KUKA KRL program: EPS_2_251455_MH12A_A_20251003045058.src

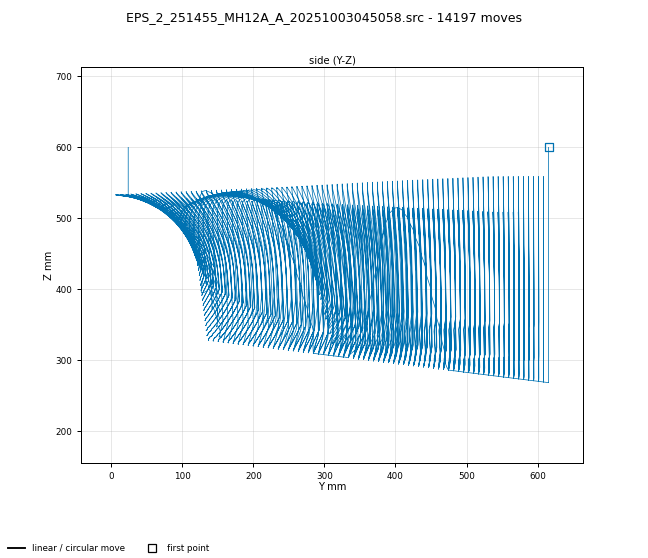
[picture p0: tool path of EPS_2_251455_MH12A_A_20251003045058.src, 14197 of 14199 moves have a stored position in this frame; points joined in program order, loops and branches not executed]
&ACCESS RVP
&REL 4
&COMMENT QRS 19112012
&PARAM EDITMASK = *
DEF PART()
EXT BAS (BAS_COMMAND :IN,REAL :IN )
INT I
BAS (#INITMOV,0 )

;KUKA QRS Post kuka4.cps  Date:22-06-2017 !

File_ID=2868

QRS_PRE_INIT()

;Init var - Until changes are made in qrs_pre_init
Outlet_Square_prg=0
Inlet_1_Square_prg=0
Inlet_2_Square_prg=0
Inlet_3_Square_prg=0
Inlet_4_Square_prg=0
Inlet_5_Square_prg=0

Outlet_1={X 0.000, Y 535.490, Z 458.500, B 0.000, E1 0.000 }
Inlet_1={X 0.000, Y 539.060, Z 408.500, B 0.000, E1 180.000 }
Inlet_2={X 0.000, Y 539.060, Z 408.500, B 0.000, E1 270.000 }
Outlet_1_type=201
Inlet_1_type=201
Inlet_2_type=201
;QRS#1=Sidecore dimensions
;QRS#2=200-8" PVC SDR 35
;QRS#3=200-8" PVC SDR 35
;QRS#4=200-8" PVC SDR 35
;QRS#5=
;QRS#6=
;QRS#7=
;QRS#8=
;QRS#9=12-08 PSX
;QRS#10=12-08 PSX
;QRS#11=12-08 PSX
;QRS#12=
;QRS#13=
;QRS#14=
;QRS#15=
;QRS#16=1220x127x838 2,75'
;QRS#17=EPS Height
;QRS#18=559
;QRS#19=*
;QRS#20= UPDATED VERSION 22-06-2017
;QRS#21=*
Outlet_Square=0100
Inlet_1_Square=0100
Inlet_2_Square=0100
Inlet_3_Square=0
Inlet_4_Square=0
Inlet_5_Square=0
Mill_Square=1
Outlet_Square_Prg=204
Inlet_1_Square_prg=204
Inlet_2_Square_prg=204

QRS_INIT()

$ADVANCE=5

; T1
PTP {E1 173.612,E2 173.612}
PTP {X 0,Y 615.502,A -85,B 0,C 180,E1 173.612,E2 173.612,E3 0,E4 0,E5 0,E6 0}
QRS_SPEED_INIT()
LIN {X 0,Y 615.502,Z 600,A -85,B 0,C 180,E1 173.612,E2 173.612,E3 0,E4 0,E5 0,E6 0} C_VEL
LIN {X 0,Y 615.502,Z 278.875,A -85,B 0,C 180,E1 173.612,E2 173.612} C_VEL
LIN {X 0,Y 615.502,Z 270.697,A -85,B 0,C 180,E1 173.612,E2 173.612} C_VEL
LIN {X 0,Y 615.472,Z 268.697,A -85,B 0,C 180,E1 173.426,E2 173.426} C_VEL
LIN {X 0,Y 615.422,Z 268.698,A -85,B 0,C 180,E1 170.8,E2 170.8} C_VEL
LIN {X 0,Y 615.459,Z 268.699,A -85,B 0,C 180,E1 168.139,E2 168.139} C_VEL
LIN {X 0,Y 615.46,Z 268.695,A -85,B 0,C 180,E1 165.45,E2 165.45} C_VEL
LIN {X 0,Y 615.453,Z 268.695,A -85,B 0,C 180,E1 163.412,E2 163.412} C_VEL
LIN {X 0,Y 615.446,Z 268.695,A -85,B 0,C 180,E1 161.353,E2 161.353} C_VEL
LIN {X 0,Y 615.437,Z 268.695,A -85,B 0,C 180,E1 159.267,E2 159.267} C_VEL
LIN {X 0,Y 615.434,Z 268.695,A -85,B 0,C 180,E1 157.153,E2 157.153} C_VEL
LIN {X 0,Y 615.433,Z 268.696,A -85,B 0,C 180,E1 155.006,E2 155.006} C_VEL
LIN {X 0,Y 615.493,Z 268.695,A -85,B 0,C 180,E1 152.085,E2 152.085} C_VEL
LIN {X 0,Y 615.478,Z 268.69,A -85,B 0,C 180,E1 149.839,E2 149.839} C_VEL
LIN {X 0,Y 615.448,Z 268.692,A -85,B 0,C 180,E1 147.54,E2 147.54} C_VEL
LIN {X 0,Y 615.44,Z 268.695,A -85,B 0,C 180,E1 145.182,E2 145.182} C_VEL
LIN {X 0,Y 615.469,Z 268.698,A -85,B 0,C 180,E1 142.756,E2 142.756} C_VEL
LIN {X 0,Y 615.47,Z 268.689,A -85,B 0,C 180,E1 139.912,E2 139.912} C_VEL
LIN {X 0,Y 615.449,Z 268.692,A -85,B 0,C 180,E1 137.643,E2 137.643} C_VEL
LIN {X 0,Y 615.469,Z 268.699,A -85,B 0,C 180,E1 134.929,E2 134.929} C_VEL
LIN {X 0,Y 615.475,Z 268.688,A -85,B 0,C 180,E1 132.079,E2 132.079} C_VEL
LIN {X 0,Y 615.452,Z 268.691,A -85,B 0,C 180,E1 129.752,E2 129.752} C_VEL
LIN {X 0,Y 615.485,Z 268.703,A -85,B 0,C 180,E1 126.936,E2 126.936} C_VEL
LIN {X 0,Y 615.459,Z 268.689,A -85,B 0,C 180,E1 124.023,E2 124.023} C_VEL
LIN {X 0,Y 615.455,Z 268.693,A -85,B 0,C 180,E1 121.686,E2 121.686} C_VEL
LIN {X 0,Y 615.47,Z 268.697,A -85,B 0,C 180,E1 119.406,E2 119.406} C_VEL
LIN {X 0,Y 615.482,Z 268.685,A -85,B 0,C 180,E1 116.443,E2 116.443} C_VEL
LIN {X 0,Y 615.46,Z 268.69,A -85,B 0,C 180,E1 114.002,E2 114.002} C_VEL
LIN {X 0,Y 615.486,Z 268.699,A -85,B 0,C 180,E1 111.431,E2 111.431} C_VEL
LIN {X 0,Y 615.486,Z 268.684,A -85,B 0,C 180,E1 108.603,E2 108.603} C_VEL
LIN {X 0,Y 615.464,Z 268.876,A -85,B 0,C 180,E1 107.957,E2 107.957} C_VEL
LIN {X 0,Y 615.478,Z 284.471,A -85,B 0,C 180,E1 105.225,E2 105.225} C_VEL
LIN {X 0,Y 615.49,Z 298.338,A -85,B 0,C 180,E1 102.823,E2 102.823} C_VEL
LIN {X 0,Y 615.481,Z 405.834,A -85,B 0,C 180,E1 101.526,E2 101.526} C_VEL
LIN {X 0,Y 615.475,Z 418.769,A -85,B 0,C 180,E1 101.234,E2 101.234} C_VEL
LIN {X 0,Y 615.492,Z 430.613,A -85,B 0,C 180,E1 100.842,E2 100.842} C_VEL
LIN {X 0,Y 615.48,Z 441.583,A -85,B 0,C 180,E1 100.36,E2 100.36} C_VEL
LIN {X 0,Y 615.493,Z 453.315,A -85,B 0,C 180,E1 99.695,E2 99.695} C_VEL
LIN {X 0,Y 615.499,Z 463.777,A -85,B 0,C 180,E1 98.949,E2 98.949} C_VEL
LIN {X 0,Y 615.498,Z 472.338,A -85,B 0,C 180,E1 98.205,E2 98.205} C_VEL
LIN {X 0,Y 615.497,Z 480.215,A -85,B 0,C 180,E1 97.38,E2 97.38} C_VEL
LIN {X 0,Y 615.497,Z 487.903,A -85,B 0,C 180,E1 96.391,E2 96.391} C_VEL
LIN {X 0,Y 615.497,Z 494.962,A -85,B 0,C 180,E1 95.24,E2 95.24} C_VEL
LIN {X 0,Y 615.494,Z 499.661,A -85,B 0,C 180,E1 94.256,E2 94.256} C_VEL
LIN {X 0,Y 615.494,Z 503.257,A -85,B 0,C 180,E1 93.272,E2 93.272} C_VEL
LIN {X 0,Y 615.496,Z 505.116,A -85,B 0,C 180,E1 92.617,E2 92.617} C_VEL
LIN {X 0,Y 615.5,Z 506.534,A -85,B 0,C 180,E1 91.962,E2 91.962} C_VEL
LIN {X 0,Y 615.496,Z 508.142,A -85,B 0,C 180,E1 90.654,E2 90.654} C_VEL
LIN {X 0,Y 615.495,Z 508.384,A -85,B 0,C 180,E1 89.999,E2 89.999} C_VEL
LIN {X 0,Y 615.495,Z 508.205,A -85,B 0,C 180,E1 89.345,E2 89.345} C_VEL
LIN {X 0,Y 615.5,Z 506.681,A -85,B 0,C 180,E1 88.036,E2 88.036} C_VEL
LIN {X 0,Y 615.498,Z 505.34,A -85,B 0,C 180,E1 87.382,E2 87.382} C_VEL
LIN {X 0,Y 615.496,Z 502.492,A -85,B 0,C 180,E1 86.399,E2 86.399} C_VEL
LIN {X 0,Y 615.498,Z 498.632,A -85,B 0,C 180,E1 85.415,E2 85.415} C_VEL
LIN {X 0,Y 615.498,Z 493.648,A -85,B 0,C 180,E1 84.43,E2 84.43} C_VEL
LIN {X 0,Y 615.496,Z 487.208,A -85,B 0,C 180,E1 83.418,E2 83.418} C_VEL
LIN {X 0,Y 615.497,Z 479.531,A -85,B 0,C 180,E1 82.454,E2 82.454} C_VEL
LIN {X 0,Y 615.498,Z 469.752,A -85,B 0,C 180,E1 81.463,E2 81.463} C_VEL
LIN {X 0,Y 615.498,Z 459.484,A -85,B 0,C 180,E1 80.635,E2 80.635} C_VEL
LIN {X 0,Y 615.483,Z 447.921,A -85,B 0,C 180,E1 79.888,E2 79.888} C_VEL
LIN {X 0,Y 615.495,Z 436.069,A -85,B 0,C 180,E1 79.293,E2 79.293} C_VEL
LIN {X 0,Y 615.475,Z 423.143,A -85,B 0,C 180,E1 78.806,E2 78.806} C_VEL
LIN {X 0,Y 615.481,Z 410.534,A -85,B 0,C 180,E1 78.473,E2 78.473} C_VEL
LIN {X 0,Y 615.49,Z 397.384,A -85,B 0,C 180,E1 78.264,E2 78.264} C_VEL
LIN {X 0,Y 615.49,Z 298.366,A -85,B 0,C 180,E1 77.092,E2 77.092} C_VEL
LIN {X 0,Y 615.48,Z 283.028,A -85,B 0,C 180,E1 74.434,E2 74.434} C_VEL
LIN {X 0,Y 615.468,Z 268.69,A -85,B 0,C 180,E1 71.901,E2 71.901} C_VEL
LIN {X 0,Y 615.488,Z 268.684,A -85,B 0,C 180,E1 69.269,E2 69.269} C_VEL
LIN {X 0,Y 615.48,Z 268.699,A -85,B 0,C 180,E1 66.443,E2 66.443} C_VEL
LIN {X 0,Y 615.484,Z 268.683,A -85,B 0,C 180,E1 63.555,E2 63.555} C_VEL
LIN {X 0,Y 615.485,Z 268.7,A -85,B 0,C 180,E1 60.593,E2 60.593} C_VEL
LIN {X 0,Y 615.487,Z 268.683,A -85,B 0,C 180,E1 57.67,E2 57.67} C_VEL
LIN {X 0,Y 615.486,Z 268.69,A -85,B 0,C 180,E1 55.184,E2 55.184} C_VEL
LIN {X 0,Y 615.49,Z 268.7,A -85,B 0,C 180,E1 52.758,E2 52.758} C_VEL
LIN {X 0,Y 615.477,Z 268.685,A -85,B 0,C 180,E1 49.913,E2 49.913} C_VEL
LIN {X 0,Y 615.488,Z 268.702,A -85,B 0,C 180,E1 46.953,E2 46.953} C_VEL
LIN {X 0,Y 615.47,Z 268.687,A -85,B 0,C 180,E1 44.151,E2 44.151} C_VEL
LIN {X 0,Y 615.484,Z 268.689,A -85,B 0,C 180,E1 41.474,E2 41.474} C_VEL
LIN {X 0,Y 615.486,Z 268.698,A -85,B 0,C 180,E1 38.905,E2 38.905} C_VEL
LIN {X 0,Y 615.468,Z 268.689,A -85,B 0,C 180,E1 36.426,E2 36.426} C_VEL
LIN {X 0,Y 615.486,Z 268.691,A -85,B 0,C 180,E1 33.533,E2 33.533} C_VEL
LIN {X 0,Y 615.474,Z 268.696,A -85,B 0,C 180,E1 30.921,E2 30.921} C_VEL
LIN {X 0,Y 615.47,Z 268.687,A -85,B 0,C 180,E1 28.447,E2 28.447} C_VEL
LIN {X 0,Y 615.487,Z 268.693,A -85,B 0,C 180,E1 25.568,E2 25.568} C_VEL
LIN {X 0,Y 615.467,Z 268.693,A -85,B 0,C 180,E1 22.845,E2 22.845} C_VEL
LIN {X 0,Y 615.492,Z 268.684,A -85,B 0,C 180,E1 20.033,E2 20.033} C_VEL
LIN {X 0,Y 615.484,Z 268.869,A -85,B 0,C 180,E1 17.957,E2 17.957} C_VEL
LIN {X 0,Y 615.454,Z 284.469,A -85,B 0,C 180,E1 15.227,E2 15.227} C_VEL
LIN {X 0,Y 615.478,Z 298.626,A -85,B 0,C 180,E1 12.803,E2 12.803} C_VEL
LIN {X 0,Y 615.484,Z 404.641,A -85,B 0,C 180,E1 11.548,E2 11.548} C_VEL
LIN {X 0,Y 615.493,Z 417.22,A -85,B 0,C 180,E1 11.276,E2 11.276} C_VEL
LIN {X 0,Y 615.493,Z 430.577,A -85,B 0,C 180,E1 10.843,E2 10.843} C_VEL
LIN {X 0,Y 615.492,Z 441.564,A -85,B 0,C 180,E1 10.361,E2 10.361} C_VEL
LIN {X 0,Y 615.479,Z 453.305,A -85,B 0,C 180,E1 9.696,E2 9.696} C_VEL
LIN {X 0,Y 615.499,Z 463.767,A -85,B 0,C 180,E1 8.95,E2 8.95} C_VEL
LIN {X 0,Y 615.498,Z 472.33,A -85,B 0,C 180,E1 8.206,E2 8.206} C_VEL
LIN {X 0,Y 615.497,Z 480.209,A -85,B 0,C 180,E1 7.38,E2 7.38} C_VEL
LIN {X 0,Y 615.497,Z 487.898,A -85,B 0,C 180,E1 6.392,E2 6.392} C_VEL
LIN {X 0,Y 615.498,Z 494.958,A -85,B 0,C 180,E1 5.241,E2 5.241} C_VEL
LIN {X 0,Y 615.493,Z 499.658,A -85,B 0,C 180,E1 4.256,E2 4.256} C_VEL
LIN {X 0,Y 615.496,Z 503.254,A -85,B 0,C 180,E1 3.273,E2 3.273} C_VEL
LIN {X 0,Y 615.496,Z 505.115,A -85,B 0,C 180,E1 2.618,E2 2.618} C_VEL
LIN {X 0,Y 615.497,Z 506.533,A -85,B 0,C 180,E1 1.963,E2 1.963} C_VEL
LIN {X 0,Y 615.496,Z 508.141,A -85,B 0,C 180,E1 0.654,E2 0.654} C_VEL
LIN {X 0,Y 615.494,Z 508.384,A -85,B 0,C 180,E1 0,E2 0} C_VEL
LIN {X 0,Y 615.496,Z 508.205,A -85,B 0,C 180,E1 -0.654,E2 -0.654} C_VEL
LIN {X 0,Y 615.496,Z 506.683,A -85,B 0,C 180,E1 -1.963,E2 -1.963} C_VEL
LIN {X 0,Y 615.498,Z 505.341,A -85,B 0,C 180,E1 -2.618,E2 -2.618} C_VEL
LIN {X 0,Y 615.496,Z 502.494,A -85,B 0,C 180,E1 -3.601,E2 -3.601} C_VEL
LIN {X 0,Y 615.499,Z 498.634,A -85,B 0,C 180,E1 -4.584,E2 -4.584} C_VEL
LIN {X 0,Y 615.498,Z 493.651,A -85,B 0,C 180,E1 -5.57,E2 -5.57} C_VEL
LIN {X 0,Y 615.497,Z 487.205,A -85,B 0,C 180,E1 -6.583,E2 -6.583} C_VEL
LIN {X 0,Y 615.497,Z 479.537,A -85,B 0,C 180,E1 -7.545,E2 -7.545} C_VEL
LIN {X 0,Y 615.498,Z 469.759,A -85,B 0,C 180,E1 -8.536,E2 -8.536} C_VEL
LIN {X 0,Y 615.497,Z 459.493,A -85,B 0,C 180,E1 -9.364,E2 -9.364} C_VEL
LIN {X 0,Y 615.487,Z 447.93,A -85,B 0,C 180,E1 -10.111,E2 -10.111} C_VEL
LIN {X 0,Y 615.498,Z 436.04,A -85,B 0,C 180,E1 -10.708,E2 -10.708} C_VEL
LIN {X 0,Y 615.492,Z 423.158,A -85,B 0,C 180,E1 -11.193,E2 -11.193} C_VEL
LIN {X 0,Y 615.485,Z 410.558,A -85,B 0,C 180,E1 -11.527,E2 -11.527} C_VEL
LIN {X 0,Y 615.478,Z 397.436,A -85,B 0,C 180,E1 -11.736,E2 -11.736} C_VEL
LIN {X 0,Y 615.485,Z 298.37,A -85,B 0,C 180,E1 -12.907,E2 -12.907} C_VEL
LIN {X 0,Y 615.492,Z 283.03,A -85,B 0,C 180,E1 -15.565,E2 -15.565} C_VEL
LIN {X 0,Y 615.44,Z 268.697,A -85,B 0,C 180,E1 -18.096,E2 -18.096} C_VEL
LIN {X 0,Y 615.438,Z 268.695,A -85,B 0,C 180,E1 -20.544,E2 -20.544} C_VEL
LIN {X 0,Y 615.464,Z 268.694,A -85,B 0,C 180,E1 -22.846,E2 -22.846} C_VEL
LIN {X 0,Y 615.441,Z 268.699,A -85,B 0,C 180,E1 -25.718,E2 -25.718} C_VEL
LIN {X 0,Y 615.424,Z 268.699,A -85,B 0,C 180,E1 -27.918,E2 -27.918} C_VEL
LIN {X 0,Y 615.42,Z 268.699,A -85,B 0,C 180,E1 -30.164,E2 -30.164} C_VEL
LIN {X 0,Y 615.434,Z 268.7,A -85,B 0,C 180,E1 -32.461,E2 -32.461} C_VEL
LIN {X 0,Y 615.482,Z 268.701,A -85,B 0,C 180,E1 -34.816,E2 -34.816} C_VEL
LIN {X 0,Y 615.449,Z 268.699,A -85,B 0,C 180,E1 -37.245,E2 -37.245} C_VEL
LIN {X 0,Y 615.42,Z 268.698,A -85,B 0,C 180,E1 -39.756,E2 -39.756} C_VEL
LIN {X 0,Y 615.46,Z 268.699,A -85,B 0,C 180,E1 -42.356,E2 -42.356} C_VEL
LIN {X 0,Y 615.458,Z 268.695,A -85,B 0,C 180,E1 -45.072,E2 -45.072} C_VEL
LIN {X 0,Y 615.432,Z 268.696,A -85,B 0,C 180,E1 -47.642,E2 -47.642} C_VEL
LIN {X 0,Y 615.483,Z 268.699,A -85,B 0,C 180,E1 -50.249,E2 -50.249} C_VEL
LIN {X 0,Y 615.452,Z 268.692,A -85,B 0,C 180,E1 -53.068,E2 -53.068} C_VEL
LIN {X 0,Y 615.442,Z 268.694,A -85,B 0,C 180,E1 -55.306,E2 -55.306} C_VEL
LIN {X 0,Y 615.456,Z 268.697,A -85,B 0,C 180,E1 -57.674,E2 -57.674} C_VEL
LIN {X 0,Y 615.487,Z 268.687,A -85,B 0,C 180,E1 -60.593,E2 -60.593} C_VEL
LIN {X 0,Y 615.456,Z 268.69,A -85,B 0,C 180,E1 -62.961,E2 -62.961} C_VEL
LIN {X 0,Y 615.455,Z 268.691,A -85,B 0,C 180,E1 -65.006,E2 -65.006} C_VEL
LIN {X 0,Y 615.456,Z 268.818,A -85,B 0,C 180,E1 -67.065,E2 -67.065} C_VEL
LIN {X 0,Y 615.471,Z 288.766,A -85,B 0,C 180,E1 -69.706,E2 -69.706} C_VEL
LIN {X 0,Y 615.492,Z 309.339,A -85,B 0,C 180,E1 -72.386,E2 -72.386} C_VEL
LIN {X 0,Y 615.494,Z 331.885,A -85,B 0,C 180,E1 -75.281,E2 -75.281} C_VEL
LIN {X 0,Y 615.491,Z 346.291,A -85,B 0,C 180,E1 -77.113,E2 -77.113} C_VEL
LIN {X 0,Y 615.484,Z 454.797,A -85,B 0,C 180,E1 -78.41,E2 -78.41} C_VEL
LIN {X 0,Y 615.475,Z 467.324,A -85,B 0,C 180,E1 -78.681,E2 -78.681} C_VEL
LIN {X 0,Y 615.489,Z 480.597,A -85,B 0,C 180,E1 -79.112,E2 -79.112} C_VEL
LIN {X 0,Y 615.48,Z 492.466,A -85,B 0,C 180,E1 -79.639,E2 -79.639} C_VEL
LIN {X 0,Y 615.493,Z 503.985,A -85,B 0,C 180,E1 -80.303,E2 -80.303} C_VEL
LIN {X 0,Y 615.499,Z 514.333,A -85,B 0,C 180,E1 -81.049,E2 -81.049} C_VEL
LIN {X 0,Y 615.497,Z 522.805,A -85,B 0,C 180,E1 -81.794,E2 -81.794} C_VEL
LIN {X 0,Y 615.498,Z 530.601,A -85,B 0,C 180,E1 -82.619,E2 -82.619} C_VEL
LIN {X 0,Y 615.496,Z 538.199,A -85,B 0,C 180,E1 -83.607,E2 -83.607} C_VEL
LIN {X 0,Y 615.498,Z 545.201,A -85,B 0,C 180,E1 -84.758,E2 -84.758} C_VEL
LIN {X 0,Y 615.493,Z 549.849,A -85,B 0,C 180,E1 -85.743,E2 -85.743} C_VEL
LIN {X 0,Y 615.495,Z 553.397,A -85,B 0,C 180,E1 -86.726,E2 -86.726} C_VEL
LIN {X 0,Y 615.497,Z 555.231,A -85,B 0,C 180,E1 -87.382,E2 -87.382} C_VEL
LIN {X 0,Y 615.499,Z 556.606,A -85,B 0,C 180,E1 -88.036,E2 -88.036} C_VEL
LIN {X 0,Y 615.496,Z 558.173,A -85,B 0,C 180,E1 -89.345,E2 -89.345} C_VEL
LIN {X 0,Y 615.494,Z 558.389,A -85,B 0,C 180,E1 -89.999,E2 -89.999} C_VEL
LIN {X 0,Y 615.496,Z 557.581,A -85,B 0,C 180,E1 -91.308,E2 -91.308} C_VEL
LIN {X 0,Y 615.499,Z 556.609,A -85,B 0,C 180,E1 -91.962,E2 -91.962} C_VEL
LIN {X 0,Y 615.497,Z 555.235,A -85,B 0,C 180,E1 -92.617,E2 -92.617} C_VEL
LIN {X 0,Y 615.496,Z 552.352,A -85,B 0,C 180,E1 -93.6,E2 -93.6} C_VEL
LIN {X 0,Y 615.498,Z 548.444,A -85,B 0,C 180,E1 -94.584,E2 -94.584} C_VEL
LIN {X 0,Y 615.499,Z 543.409,A -85,B 0,C 180,E1 -95.569,E2 -95.569} C_VEL
LIN {X 0,Y 615.497,Z 536.87,A -85,B 0,C 180,E1 -96.583,E2 -96.583} C_VEL
LIN {X 0,Y 615.497,Z 529.139,A -85,B 0,C 180,E1 -97.545,E2 -97.545} C_VEL
LIN {X 0,Y 615.498,Z 521.053,A -85,B 0,C 180,E1 -98.37,E2 -98.37} C_VEL
LIN {X 0,Y 615.499,Z 511.177,A -85,B 0,C 180,E1 -99.198,E2 -99.198} C_VEL
LIN {X 0,Y 615.492,Z 499.993,A -85,B 0,C 180,E1 -99.944,E2 -99.944} C_VEL
LIN {X 0,Y 615.485,Z 489.038,A -85,B 0,C 180,E1 -100.526,E2 -100.526} C_VEL
LIN {X 0,Y 615.48,Z 476.491,A -85,B 0,C 180,E1 -101.04,E2 -101.04} C_VEL
LIN {X 0,Y 615.476,Z 464.1,A -85,B 0,C 180,E1 -101.401,E2 -101.401} C_VEL
LIN {X 0,Y 615.488,Z 450.519,A -85,B 0,C 180,E1 -101.651,E2 -101.651} C_VEL
LIN {X 0,Y 615.491,Z 346.302,A -85,B 0,C 180,E1 -102.886,E2 -102.886} C_VEL
LIN {X 0,Y 615.497,Z 323.939,A -85,B 0,C 180,E1 -105.734,E2 -105.734} C_VEL
LIN {X 0,Y 615.49,Z 301.384,A -85,B 0,C 180,E1 -108.645,E2 -108.645} C_VEL
LIN {X 0,Y 615.489,Z 278.801,A -85,B 0,C 180,E1 -111.607,E2 -111.607} C_VEL
LIN {X 0,Y 615.456,Z 268.691,A -85,B 0,C 180,E1 -112.978,E2 -112.978} C_VEL
LIN {X 0,Y 615.493,Z 268.688,A -85,B 0,C 180,E1 -115.715,E2 -115.715} C_VEL
LIN {X 0,Y 615.454,Z 268.694,A -85,B 0,C 180,E1 -118.659,E2 -118.659} C_VEL
LIN {X 0,Y 615.462,Z 268.689,A -85,B 0,C 180,E1 -121.082,E2 -121.082} C_VEL
LIN {X 0,Y 615.484,Z 268.7,A -85,B 0,C 180,E1 -124.021,E2 -124.021} C_VEL
LIN {X 0,Y 615.451,Z 268.695,A -85,B 0,C 180,E1 -126.426,E2 -126.426} C_VEL
LIN {X 0,Y 615.468,Z 268.689,A -85,B 0,C 180,E1 -129.06,E2 -129.06} C_VEL
LIN {X 0,Y 615.459,Z 268.698,A -85,B 0,C 180,E1 -132.077,E2 -132.077} C_VEL
LIN {X 0,Y 615.451,Z 268.696,A -85,B 0,C 180,E1 -134.152,E2 -134.152} C_VEL
LIN {X 0,Y 615.468,Z 268.69,A -85,B 0,C 180,E1 -136.953,E2 -136.953} C_VEL
LIN {X 0,Y 615.455,Z 268.697,A -85,B 0,C 180,E1 -139.913,E2 -139.913} C_VEL
LIN {X 0,Y 615.442,Z 268.698,A -85,B 0,C 180,E1 -141.992,E2 -141.992} C_VEL
LIN {X 0,Y 615.437,Z 268.694,A -85,B 0,C 180,E1 -144.381,E2 -144.381} C_VEL
LIN {X 0,Y 615.463,Z 268.692,A -85,B 0,C 180,E1 -146.762,E2 -146.762} C_VEL
LIN {X 0,Y 615.491,Z 268.695,A -85,B 0,C 180,E1 -149.08,E2 -149.08} C_VEL
LIN {X 0,Y 615.457,Z 268.699,A -85,B 0,C 180,E1 -151.553,E2 -151.553} C_VEL
LIN {X 0,Y 615.45,Z 268.699,A -85,B 0,C 180,E1 -153.554,E2 -153.554} C_VEL
LIN {X 0,Y 615.427,Z 268.697,A -85,B 0,C 180,E1 -156.002,E2 -156.002} C_VEL
LIN {X 0,Y 615.456,Z 268.696,A -85,B 0,C 180,E1 -158.567,E2 -158.567} C_VEL
LIN {X 0,Y 615.444,Z 268.699,A -85,B 0,C 180,E1 -161.404,E2 -161.404} C_VEL
LIN {X 0,Y 615.427,Z 268.698,A -85,B 0,C 180,E1 -163.585,E2 -163.585} C_VEL
LIN {X 0,Y 615.429,Z 268.699,A -85,B 0,C 180,E1 -165.449,E2 -165.449} C_VEL
LIN {X 0,Y 615.426,Z 268.699,A -85,B 0,C 180,E1 -167.469,E2 -167.469} C_VEL
LIN {X 0,Y 615.422,Z 268.699,A -85,B 0,C 180,E1 -169.472,E2 -169.472} C_VEL
LIN {X 0,Y 615.419,Z 268.699,A -85,B 0,C 180,E1 -171.462,E2 -171.462} C_VEL
LIN {X 0,Y 615.416,Z 268.7,A -85,B 0,C 180,E1 -173.471,E2 -173.471} C_VEL
LIN {X 0,Y 615.414,Z 268.7,A -85,B 0,C 180,E1 -175.415,E2 -175.415} C_VEL
LIN {X 0,Y 615.414,Z 268.7,A -85,B 0,C 180,E1 -177.382,E2 -177.382} C_VEL
LIN {X 0,Y 615.415,Z 268.7,A -85,B 0,C 180,E1 -179.346,E2 -179.346} C_VEL
LIN {X 0,Y 615.417,Z 268.699,A -85,B 0,C 180,E1 -181.309,E2 -181.309} C_VEL
LIN {X 0,Y 615.416,Z 268.699,A -85,B 0,C 180,E1 -183.273,E2 -183.273} C_VEL
LIN {X 0,Y 615.42,Z 268.698,A -85,B 0,C 180,E1 -185.242,E2 -185.242} C_VEL
LIN {X 0,Y 615.472,Z 268.697,A -85,B 0,C 180,E1 -186.574,E2 -186.574} C_VEL
LIN {X 0,Y 614.761,Z 268.842,A -85,B 0,C 180,E1 -187.12,E2 -187.12} C_VEL
LIN {X 0,Y 611.901,Z 269.264,A -85,B 0,C 180,E1 -188.006,E2 -188.006} C_VEL
LIN {X 0,Y 609.514,Z 269.569,A -85,B 0,C 180,E1 -188.718,E2 -188.718} C_VEL
LIN {X 0,Y 608.493,Z 269.684,A -85,B 0,C 180,E1 -189.268,E2 -189.268} C_VEL
LIN {X 0,Y 608.41,Z 269.693,A -85,B 0,C 180,E1 -189.454,E2 -189.454} C_VEL
LIN {X 0,Y 608.438,Z 269.697,A -85,B 0,C 180,E1 -192,E2 -192} C_VEL
LIN {X 0,Y 608.415,Z 269.694,A -85,B 0,C 180,E1 -194.722,E2 -194.722} C_VEL
LIN {X 0,Y 608.414,Z 269.693,A -85,B 0,C 180,E1 -196.785,E2 -196.785} C_VEL
LIN {X 0,Y 608.423,Z 269.695,A -85,B 0,C 180,E1 -199.572,E2 -199.572} C_VEL
LIN {X 0,Y 608.451,Z 269.69,A -85,B 0,C 180,E1 -202.477,E2 -202.477} C_VEL
LIN {X 0,Y 608.428,Z 269.691,A -85,B 0,C 180,E1 -204.572,E2 -204.572} C_VEL
LIN {X 0,Y 608.44,Z 269.691,A -85,B 0,C 180,E1 -207.202,E2 -207.202} C_VEL
LIN {X 0,Y 608.47,Z 269.691,A -85,B 0,C 180,E1 -209.974,E2 -209.974} C_VEL
LIN {X 0,Y 608.43,Z 269.691,A -85,B 0,C 180,E1 -212.881,E2 -212.881} C_VEL
LIN {X 0,Y 608.432,Z 269.696,A -85,B 0,C 180,E1 -215.279,E2 -215.279} C_VEL
LIN {X 0,Y 608.451,Z 269.688,A -85,B 0,C 180,E1 -218.24,E2 -218.24} C_VEL
LIN {X 0,Y 608.459,Z 269.697,A -85,B 0,C 180,E1 -221.343,E2 -221.343} C_VEL
LIN {X 0,Y 608.459,Z 269.689,A -85,B 0,C 180,E1 -223.871,E2 -223.871} C_VEL
LIN {X 0,Y 608.446,Z 269.691,A -85,B 0,C 180,E1 -226.694,E2 -226.694} C_VEL
LIN {X 0,Y 608.433,Z 269.694,A -85,B 0,C 180,E1 -228.823,E2 -228.823} C_VEL
LIN {X 0,Y 608.455,Z 269.689,A -85,B 0,C 180,E1 -231.762,E2 -231.762} C_VEL
LIN {X 0,Y 608.437,Z 269.69,A -85,B 0,C 180,E1 -233.956,E2 -233.956} C_VEL
LIN {X 0,Y 608.44,Z 269.69,A -85,B 0,C 180,E1 -236.329,E2 -236.329} C_VEL
LIN {X 0,Y 608.442,Z 269.696,A -85,B 0,C 180,E1 -238.734,E2 -238.734} C_VEL
LIN {X 0,Y 608.474,Z 269.688,A -85,B 0,C 180,E1 -241.38,E2 -241.38} C_VEL
LIN {X 0,Y 608.431,Z 269.691,A -85,B 0,C 180,E1 -243.965,E2 -243.965} C_VEL
LIN {X 0,Y 608.446,Z 269.69,A -85,B 0,C 180,E1 -246.155,E2 -246.155} C_VEL
LIN {X 0,Y 608.458,Z 269.692,A -85,B 0,C 180,E1 -249.019,E2 -249.019} C_VEL
LIN {X 0,Y 608.44,Z 269.696,A -85,B 0,C 180,E1 -251.959,E2 -251.959} C_VEL
LIN {X 0,Y 608.474,Z 284.61,A -85,B 0,C 180,E1 -254.595,E2 -254.595} C_VEL
LIN {X 0,Y 608.488,Z 298.779,A -85,B 0,C 180,E1 -257.048,E2 -257.048} C_VEL
LIN {X 0,Y 608.55,Z 404.834,A -85,B 0,C 180,E1 -258.32,E2 -258.32} C_VEL
LIN {X 0,Y 608.523,Z 418.149,A -85,B 0,C 180,E1 -258.615,E2 -258.615} C_VEL
LIN {X 0,Y 608.526,Z 431.388,A -85,B 0,C 180,E1 -259.056,E2 -259.056} C_VEL
LIN {X 0,Y 608.491,Z 443.385,A -85,B 0,C 180,E1 -259.604,E2 -259.604} C_VEL
LIN {X 0,Y 608.507,Z 454.802,A -85,B 0,C 180,E1 -260.276,E2 -260.276} C_VEL
LIN {X 0,Y 608.474,Z 465.094,A -85,B 0,C 180,E1 -261.03,E2 -261.03} C_VEL
LIN {X 0,Y 608.463,Z 474.358,A -85,B 0,C 180,E1 -261.867,E2 -261.867} C_VEL
LIN {X 0,Y 608.466,Z 483.33,A -85,B 0,C 180,E1 -262.868,E2 -262.868} C_VEL
LIN {X 0,Y 608.444,Z 490.56,A -85,B 0,C 180,E1 -263.867,E2 -263.867} C_VEL
LIN {X 0,Y 608.462,Z 495.439,A -85,B 0,C 180,E1 -264.699,E2 -264.699} C_VEL
LIN {X 0,Y 608.439,Z 500.182,A -85,B 0,C 180,E1 -265.695,E2 -265.695} C_VEL
LIN {X 0,Y 608.425,Z 503.814,A -85,B 0,C 180,E1 -266.69,E2 -266.69} C_VEL
LIN {X 0,Y 608.425,Z 505.692,A -85,B 0,C 180,E1 -267.352,E2 -267.352} C_VEL
LIN {X 0,Y 608.444,Z 507.128,A -85,B 0,C 180,E1 -268.015,E2 -268.015} C_VEL
LIN {X 0,Y 608.439,Z 508.752,A -85,B 0,C 180,E1 -269.339,E2 -269.339} C_VEL
LIN {X 0,Y 608.435,Z 508.996,A -85,B 0,C 180,E1 -270.001,E2 -270.001} C_VEL
LIN {X 0,Y 608.438,Z 508.815,A -85,B 0,C 180,E1 -270.662,E2 -270.662} C_VEL
LIN {X 0,Y 608.445,Z 507.275,A -85,B 0,C 180,E1 -271.986,E2 -271.986} C_VEL
LIN {X 0,Y 608.426,Z 505.917,A -85,B 0,C 180,E1 -272.649,E2 -272.649} C_VEL
LIN {X 0,Y 608.449,Z 503.04,A -85,B 0,C 180,E1 -273.643,E2 -273.643} C_VEL
LIN {X 0,Y 608.433,Z 499.14,A -85,B 0,C 180,E1 -274.638,E2 -274.638} C_VEL
LIN {X 0,Y 608.45,Z 494.109,A -85,B 0,C 180,E1 -275.635,E2 -275.635} C_VEL
LIN {X 0,Y 608.441,Z 487.79,A -85,B 0,C 180,E1 -276.634,E2 -276.634} C_VEL
LIN {X 0,Y 608.476,Z 479.874,A -85,B 0,C 180,E1 -277.634,E2 -277.634} C_VEL
LIN {X 0,Y 608.472,Z 470.03,A -85,B 0,C 180,E1 -278.636,E2 -278.636} C_VEL
LIN {X 0,Y 608.48,Z 459.706,A -85,B 0,C 180,E1 -279.474,E2 -279.474} C_VEL
LIN {X 0,Y 608.479,Z 448.092,A -85,B 0,C 180,E1 -280.23,E2 -280.23} C_VEL
LIN {X 0,Y 608.51,Z 436.204,A -85,B 0,C 180,E1 -280.831,E2 -280.831} C_VEL
LIN {X 0,Y 608.519,Z 423.248,A -85,B 0,C 180,E1 -281.324,E2 -281.324} C_VEL
LIN {X 0,Y 608.541,Z 410.626,A -85,B 0,C 180,E1 -281.661,E2 -281.661} C_VEL
LIN {X 0,Y 608.544,Z 397.49,A -85,B 0,C 180,E1 -281.872,E2 -281.872} C_VEL
LIN {X 0,Y 608.522,Z 299.095,A -85,B 0,C 180,E1 -283.037,E2 -283.037} C_VEL
LIN {X 0,Y 608.463,Z 298.324,A -85,B 0,C 180,E1 -283.102,E2 -283.102} C_VEL
LIN {X 0,Y 608.459,Z 283.158,A -85,B 0,C 180,E1 -285.75,E2 -285.75} C_VEL
LIN {X 0,Y 608.454,Z 269.689,A -85,B 0,C 180,E1 -288.151,E2 -288.151} C_VEL
LIN {X 0,Y 608.463,Z 269.689,A -85,B 0,C 180,E1 -290.982,E2 -290.982} C_VEL
LIN {X 0,Y 608.452,Z 269.691,A -85,B 0,C 180,E1 -293.846,E2 -293.846} C_VEL
LIN {X 0,Y 608.447,Z 269.69,A -85,B 0,C 180,E1 -296.775,E2 -296.775} C_VEL
LIN {X 0,Y 608.471,Z 269.691,A -85,B 0,C 180,E1 -299.02,E2 -299.02} C_VEL
LIN {X 0,Y 608.463,Z 269.686,A -85,B 0,C 180,E1 -302.095,E2 -302.095} C_VEL
LIN {X 0,Y 608.45,Z 269.693,A -85,B 0,C 180,E1 -304.905,E2 -304.905} C_VEL
LIN {X 0,Y 608.463,Z 269.688,A -85,B 0,C 180,E1 -307.747,E2 -307.747} C_VEL
LIN {X 0,Y 608.447,Z 269.689,A -85,B 0,C 180,E1 -310.328,E2 -310.328} C_VEL
LIN {X 0,Y 608.473,Z 269.691,A -85,B 0,C 180,E1 -313.309,E2 -313.309} C_VEL
LIN {X 0,Y 608.466,Z 269.686,A -85,B 0,C 180,E1 -316.13,E2 -316.13} C_VEL
LIN {X 0,Y 608.458,Z 269.695,A -85,B 0,C 180,E1 -318.823,E2 -318.823} C_VEL
LIN {X 0,Y 608.439,Z 269.692,A -85,B 0,C 180,E1 -321.41,E2 -321.41} C_VEL
LIN {X 0,Y 608.451,Z 269.688,A -85,B 0,C 180,E1 -323.955,E2 -323.955} C_VEL
LIN {X 0,Y 608.453,Z 269.69,A -85,B 0,C 180,E1 -326.328,E2 -326.328} C_VEL
LIN {X 0,Y 608.451,Z 269.697,A -85,B 0,C 180,E1 -328.732,E2 -328.732} C_VEL
LIN {X 0,Y 608.459,Z 269.688,A -85,B 0,C 180,E1 -331.383,E2 -331.383} C_VEL
LIN {X 0,Y 608.439,Z 269.69,A -85,B 0,C 180,E1 -333.964,E2 -333.964} C_VEL
LIN {X 0,Y 608.47,Z 269.688,A -85,B 0,C 180,E1 -336.155,E2 -336.155} C_VEL
LIN {X 0,Y 608.45,Z 269.692,A -85,B 0,C 180,E1 -339.018,E2 -339.018} C_VEL
LIN {X 0,Y 608.463,Z 269.691,A -85,B 0,C 180,E1 -341.959,E2 -341.959} C_VEL
LIN {X 0,Y 608.46,Z 284.605,A -85,B 0,C 180,E1 -344.594,E2 -344.594} C_VEL
LIN {X 0,Y 608.451,Z 298.708,A -85,B 0,C 180,E1 -347.047,E2 -347.047} C_VEL
LIN {X 0,Y 608.542,Z 404.777,A -85,B 0,C 180,E1 -348.319,E2 -348.319} C_VEL
LIN {X 0,Y 608.535,Z 418.12,A -85,B 0,C 180,E1 -348.614,E2 -348.614} C_VEL
LIN {X 0,Y 608.542,Z 430.175,A -85,B 0,C 180,E1 -349.011,E2 -349.011} C_VEL
LIN {X 0,Y 608.514,Z 441.724,A -85,B 0,C 180,E1 -349.519,E2 -349.519} C_VEL
LIN {X 0,Y 608.469,Z 453.513,A -85,B 0,C 180,E1 -350.191,E2 -350.191} C_VEL
LIN {X 0,Y 608.474,Z 465.084,A -85,B 0,C 180,E1 -351.029,E2 -351.029} C_VEL
LIN {X 0,Y 608.464,Z 474.348,A -85,B 0,C 180,E1 -351.866,E2 -351.866} C_VEL
LIN {X 0,Y 608.466,Z 483.323,A -85,B 0,C 180,E1 -352.867,E2 -352.867} C_VEL
LIN {X 0,Y 608.444,Z 490.556,A -85,B 0,C 180,E1 -353.866,E2 -353.866} C_VEL
LIN {X 0,Y 608.463,Z 495.435,A -85,B 0,C 180,E1 -354.698,E2 -354.698} C_VEL
LIN {X 0,Y 608.439,Z 500.179,A -85,B 0,C 180,E1 -355.694,E2 -355.694} C_VEL
LIN {X 0,Y 608.426,Z 503.813,A -85,B 0,C 180,E1 -356.689,E2 -356.689} C_VEL
LIN {X 0,Y 608.425,Z 505.69,A -85,B 0,C 180,E1 -357.352,E2 -357.352} C_VEL
LIN {X 0,Y 608.442,Z 507.126,A -85,B 0,C 180,E1 -358.014,E2 -358.014} C_VEL
LIN {X 0,Y 608.439,Z 508.752,A -85,B 0,C 180,E1 -359.338,E2 -359.338} C_VEL
LIN {X 0,Y 608.434,Z 508.995,A -85,B 0,C 180,E1 -360,E2 -360} C_VEL
LIN {X 0,Y 608.439,Z 508.815,A -85,B 0,C 180,E1 -360.662,E2 -360.662} C_VEL
LIN {X 0,Y 608.441,Z 507.276,A -85,B 0,C 180,E1 -361.986,E2 -361.986} C_VEL
LIN {X 0,Y 608.426,Z 505.919,A -85,B 0,C 180,E1 -362.648,E2 -362.648} C_VEL
LIN {X 0,Y 608.45,Z 503.042,A -85,B 0,C 180,E1 -363.642,E2 -363.642} C_VEL
LIN {X 0,Y 608.433,Z 499.144,A -85,B 0,C 180,E1 -364.638,E2 -364.638} C_VEL
LIN {X 0,Y 608.449,Z 494.113,A -85,B 0,C 180,E1 -365.634,E2 -365.634} C_VEL
LIN {X 0,Y 608.441,Z 487.791,A -85,B 0,C 180,E1 -366.633,E2 -366.633} C_VEL
LIN {X 0,Y 608.475,Z 479.879,A -85,B 0,C 180,E1 -367.633,E2 -367.633} C_VEL
LIN {X 0,Y 608.472,Z 470.037,A -85,B 0,C 180,E1 -368.636,E2 -368.636} C_VEL
LIN {X 0,Y 608.479,Z 459.709,A -85,B 0,C 180,E1 -369.473,E2 -369.473} C_VEL
LIN {X 0,Y 608.484,Z 448.09,A -85,B 0,C 180,E1 -370.229,E2 -370.229} C_VEL
LIN {X 0,Y 608.52,Z 435.875,A -85,B 0,C 180,E1 -370.845,E2 -370.845} C_VEL
LIN {X 0,Y 608.53,Z 423.256,A -85,B 0,C 180,E1 -371.323,E2 -371.323} C_VEL
LIN {X 0,Y 608.532,Z 410.629,A -85,B 0,C 180,E1 -371.66,E2 -371.66} C_VEL
LIN {X 0,Y 608.534,Z 397.539,A -85,B 0,C 180,E1 -371.872,E2 -371.872} C_VEL
LIN {X 0,Y 608.529,Z 299.143,A -85,B 0,C 180,E1 -373.036,E2 -373.036} C_VEL
LIN {X 0,Y 608.472,Z 298.327,A -85,B 0,C 180,E1 -373.101,E2 -373.101} C_VEL
LIN {X 0,Y 608.478,Z 283.161,A -85,B 0,C 180,E1 -375.749,E2 -375.749} C_VEL
LIN {X 0,Y 608.425,Z 269.693,A -85,B 0,C 180,E1 -378.151,E2 -378.151} C_VEL
LIN {X 0,Y 608.441,Z 269.693,A -85,B 0,C 180,E1 -380.982,E2 -380.982} C_VEL
LIN {X 0,Y 608.425,Z 269.693,A -85,B 0,C 180,E1 -383.847,E2 -383.847} C_VEL
LIN {X 0,Y 608.403,Z 269.694,A -85,B 0,C 180,E1 -386.038,E2 -386.038} C_VEL
LIN {X 0,Y 608.437,Z 269.692,A -85,B 0,C 180,E1 -388.613,E2 -388.613} C_VEL
LIN {X 0,Y 608.435,Z 269.695,A -85,B 0,C 180,E1 -391.318,E2 -391.318} C_VEL
LIN {X 0,Y 608.4,Z 269.695,A -85,B 0,C 180,E1 -393.724,E2 -393.724} C_VEL
LIN {X 0,Y 608.39,Z 269.696,A -85,B 0,C 180,E1 -396.096,E2 -396.096} C_VEL
LIN {X 0,Y 608.416,Z 269.699,A -85,B 0,C 180,E1 -398.592,E2 -398.592} C_VEL
LIN {X 0,Y 608.423,Z 269.693,A -85,B 0,C 180,E1 -401.337,E2 -401.337} C_VEL
LIN {X 0,Y 608.427,Z 269.692,A -85,B 0,C 180,E1 -403.874,E2 -403.874} C_VEL
LIN {X 0,Y 608.479,Z 269.691,A -85,B 0,C 180,E1 -406.691,E2 -406.691} C_VEL
LIN {X 0,Y 608.445,Z 269.693,A -85,B 0,C 180,E1 -408.822,E2 -408.822} C_VEL
LIN {X 0,Y 608.409,Z 269.693,A -85,B 0,C 180,E1 -411.407,E2 -411.407} C_VEL
LIN {X 0,Y 608.444,Z 269.694,A -85,B 0,C 180,E1 -413.955,E2 -413.955} C_VEL
LIN {X 0,Y 608.471,Z 269.693,A -85,B 0,C 180,E1 -416.329,E2 -416.329} C_VEL
LIN {X 0,Y 608.443,Z 269.69,A -85,B 0,C 180,E1 -418.733,E2 -418.733} C_VEL
LIN {X 0,Y 608.447,Z 269.69,A -85,B 0,C 180,E1 -421.385,E2 -421.385} C_VEL
LIN {X 0,Y 608.48,Z 269.689,A -85,B 0,C 180,E1 -424.278,E2 -424.278} C_VEL
LIN {X 0,Y 608.459,Z 269.816,A -85,B 0,C 180,E1 -426.921,E2 -426.921} C_VEL
LIN {X 0,Y 608.584,Z 285.438,A -85,B 0,C 180,E1 -429.023,E2 -429.023} C_VEL
LIN {X 0,Y 608.521,Z 306.712,A -85,B 0,C 180,E1 -431.83,E2 -431.83} C_VEL
LIN {X 0,Y 608.498,Z 326.656,A -85,B 0,C 180,E1 -434.423,E2 -434.423} C_VEL
LIN {X 0,Y 608.497,Z 346.517,A -85,B 0,C 180,E1 -436.973,E2 -436.973} C_VEL
LIN {X 0,Y 608.544,Z 454.914,A -85,B 0,C 180,E1 -438.276,E2 -438.276} C_VEL
LIN {X 0,Y 608.51,Z 468.193,A -85,B 0,C 180,E1 -438.571,E2 -438.571} C_VEL
LIN {X 0,Y 608.516,Z 480.606,A -85,B 0,C 180,E1 -438.981,E2 -438.981} C_VEL
LIN {X 0,Y 608.502,Z 492.623,A -85,B 0,C 180,E1 -439.519,E2 -439.519} C_VEL
LIN {X 0,Y 608.487,Z 504.188,A -85,B 0,C 180,E1 -440.191,E2 -440.191} C_VEL
LIN {X 0,Y 608.485,Z 514.586,A -85,B 0,C 180,E1 -440.945,E2 -440.945} C_VEL
LIN {X 0,Y 608.475,Z 523.105,A -85,B 0,C 180,E1 -441.698,E2 -441.698} C_VEL
LIN {X 0,Y 608.471,Z 530.955,A -85,B 0,C 180,E1 -442.533,E2 -442.533} C_VEL
LIN {X 0,Y 608.461,Z 538.284,A -85,B 0,C 180,E1 -443.484,E2 -443.484} C_VEL
LIN {X 0,Y 608.45,Z 543.862,A -85,B 0,C 180,E1 -444.365,E2 -444.365} C_VEL
LIN {X 0,Y 608.432,Z 548.947,A -85,B 0,C 180,E1 -445.362,E2 -445.362} C_VEL
LIN {X 0,Y 608.449,Z 552.894,A -85,B 0,C 180,E1 -446.357,E2 -446.357} C_VEL
LIN {X 0,Y 608.425,Z 555.807,A -85,B 0,C 180,E1 -447.351,E2 -447.351} C_VEL
LIN {X 0,Y 608.444,Z 557.2,A -85,B 0,C 180,E1 -448.014,E2 -448.014} C_VEL
LIN {X 0,Y 608.438,Z 558.783,A -85,B 0,C 180,E1 -449.338,E2 -449.338} C_VEL
LIN {X 0,Y 608.434,Z 559,A -85,B 0,C 180,E1 -449.999,E2 -449.999} C_VEL
LIN {X 0,Y 608.448,Z 558.185,A -85,B 0,C 180,E1 -451.323,E2 -451.323} C_VEL
LIN {X 0,Y 608.444,Z 557.202,A -85,B 0,C 180,E1 -451.985,E2 -451.985} C_VEL
LIN {X 0,Y 608.425,Z 555.811,A -85,B 0,C 180,E1 -452.648,E2 -452.648} C_VEL
LIN {X 0,Y 608.449,Z 552.898,A -85,B 0,C 180,E1 -453.642,E2 -453.642} C_VEL
LIN {X 0,Y 608.432,Z 548.953,A -85,B 0,C 180,E1 -454.637,E2 -454.637} C_VEL
LIN {X 0,Y 608.437,Z 542.881,A -85,B 0,C 180,E1 -455.8,E2 -455.8} C_VEL
LIN {X 0,Y 608.461,Z 536.24,A -85,B 0,C 180,E1 -456.799,E2 -456.799} C_VEL
LIN {X 0,Y 608.455,Z 527.995,A -85,B 0,C 180,E1 -457.799,E2 -457.799} C_VEL
LIN {X 0,Y 608.472,Z 519.544,A -85,B 0,C 180,E1 -458.635,E2 -458.635} C_VEL
LIN {X 0,Y 608.471,Z 509.101,A -85,B 0,C 180,E1 -459.473,E2 -459.473} C_VEL
LIN {X 0,Y 608.493,Z 498.768,A -85,B 0,C 180,E1 -460.144,E2 -460.144} C_VEL
LIN {X 0,Y 608.522,Z 487.275,A -85,B 0,C 180,E1 -460.739,E2 -460.739} C_VEL
LIN {X 0,Y 608.527,Z 474.904,A -85,B 0,C 180,E1 -461.224,E2 -461.224} C_VEL
LIN {X 0,Y 608.541,Z 461.472,A -85,B 0,C 180,E1 -461.596,E2 -461.596} C_VEL
LIN {X 0,Y 608.551,Z 449.141,A -85,B 0,C 180,E1 -461.807,E2 -461.807} C_VEL
LIN {X 0,Y 608.487,Z 346.445,A -85,B 0,C 180,E1 -463.037,E2 -463.037} C_VEL
LIN {X 0,Y 608.508,Z 324.008,A -85,B 0,C 180,E1 -465.92,E2 -465.92} C_VEL
LIN {X 0,Y 608.544,Z 302.396,A -85,B 0,C 180,E1 -468.736,E2 -468.736} C_VEL
LIN {X 0,Y 608.593,Z 280.131,A -85,B 0,C 180,E1 -471.686,E2 -471.686} C_VEL
LIN {X 0,Y 608.432,Z 269.692,A -85,B 0,C 180,E1 -473.101,E2 -473.101} C_VEL
LIN {X 0,Y 608.478,Z 269.688,A -85,B 0,C 180,E1 -475.722,E2 -475.722} C_VEL
LIN {X 0,Y 608.45,Z 269.69,A -85,B 0,C 180,E1 -478.615,E2 -478.615} C_VEL
LIN {X 0,Y 608.441,Z 269.69,A -85,B 0,C 180,E1 -481.317,E2 -481.317} C_VEL
LIN {X 0,Y 608.478,Z 269.691,A -85,B 0,C 180,E1 -483.735,E2 -483.735} C_VEL
LIN {X 0,Y 608.44,Z 269.696,A -85,B 0,C 180,E1 -486.092,E2 -486.092} C_VEL
LIN {X 0,Y 608.417,Z 269.692,A -85,B 0,C 180,E1 -488.591,E2 -488.591} C_VEL
LIN {X 0,Y 608.462,Z 269.69,A -85,B 0,C 180,E1 -491.342,E2 -491.342} C_VEL
LIN {X 0,Y 608.453,Z 269.695,A -85,B 0,C 180,E1 -493.87,E2 -493.87} C_VEL
LIN {X 0,Y 608.443,Z 269.689,A -85,B 0,C 180,E1 -496.693,E2 -496.693} C_VEL
LIN {X 0,Y 608.446,Z 269.696,A -85,B 0,C 180,E1 -499.696,E2 -499.696} C_VEL
LIN {X 0,Y 608.433,Z 269.69,A -85,B 0,C 180,E1 -502.251,E2 -502.251} C_VEL
LIN {X 0,Y 608.455,Z 269.693,A -85,B 0,C 180,E1 -505.092,E2 -505.092} C_VEL
LIN {X 0,Y 608.432,Z 269.692,A -85,B 0,C 180,E1 -507.903,E2 -507.903} C_VEL
LIN {X 0,Y 608.419,Z 269.692,A -85,B 0,C 180,E1 -510.218,E2 -510.218} C_VEL
LIN {X 0,Y 608.456,Z 269.691,A -85,B 0,C 180,E1 -512.795,E2 -512.795} C_VEL
LIN {X 0,Y 608.431,Z 269.695,A -85,B 0,C 180,E1 -515.428,E2 -515.428} C_VEL
LIN {X 0,Y 608.429,Z 269.691,A -85,B 0,C 180,E1 -518.307,E2 -518.307} C_VEL
LIN {X 0,Y 608.443,Z 269.694,A -85,B 0,C 180,E1 -521.289,E2 -521.289} C_VEL
LIN {X 0,Y 608.405,Z 269.694,A -85,B 0,C 180,E1 -523.905,E2 -523.905} C_VEL
LIN {X 0,Y 608.457,Z 269.695,A -85,B 0,C 180,E1 -526.643,E2 -526.643} C_VEL
LIN {X 0,Y 608.412,Z 269.694,A -85,B 0,C 180,E1 -529.349,E2 -529.349} C_VEL
LIN {X 0,Y 608.404,Z 269.695,A -85,B 0,C 180,E1 -531.363,E2 -531.363} C_VEL
LIN {X 0,Y 608.402,Z 269.694,A -85,B 0,C 180,E1 -533.422,E2 -533.422} C_VEL
LIN {X 0,Y 608.389,Z 269.696,A -85,B 0,C 180,E1 -535.362,E2 -535.362} C_VEL
LIN {X 0,Y 608.413,Z 269.693,A -85,B 0,C 180,E1 -537.352,E2 -537.352} C_VEL
LIN {X 0,Y 608.432,Z 269.693,A -85,B 0,C 180,E1 -540,E2 -540} C_VEL
LIN {X 0,Y 608.463,Z 269.693,A -85,B 0,C 180,E1 -542.648,E2 -542.648} C_VEL
LIN {X 0,Y 608.404,Z 269.694,A -85,B 0,C 180,E1 -545.302,E2 -545.302} C_VEL
LIN {X 0,Y 608.401,Z 269.694,A -85,B 0,C 180,E1 -547.3,E2 -547.3} C_VEL
LIN {X 0,Y 608.41,Z 269.693,A -85,B 0,C 180,E1 -549.454,E2 -549.454} C_VEL
LIN {X 0,Y 607.748,Z 269.784,A -85,B 0,C 180,E1 -550.007,E2 -550.007} C_VEL
LIN {X 0,Y 604.909,Z 270.141,A -85,B 0,C 180,E1 -550.904,E2 -550.904} C_VEL
LIN {X 0,Y 602.506,Z 270.441,A -85,B 0,C 180,E1 -551.625,E2 -551.625} C_VEL
LIN {X 0,Y 601.47,Z 270.568,A -85,B 0,C 180,E1 -552.182,E2 -552.182} C_VEL
LIN {X 0,Y 601.383,Z 270.574,A -85,B 0,C 180,E1 -552.371,E2 -552.371} C_VEL
LIN {X 0,Y 601.38,Z 270.569,A -85,B 0,C 180,E1 -554.898,E2 -554.898} C_VEL
LIN {X 0,Y 601.389,Z 270.568,A -85,B 0,C 180,E1 -556.987,E2 -556.987} C_VEL
LIN {X 0,Y 601.384,Z 270.576,A -85,B 0,C 180,E1 -559.81,E2 -559.81} C_VEL
LIN {X 0,Y 601.4,Z 270.567,A -85,B 0,C 180,E1 -562.684,E2 -562.684} C_VEL
LIN {X 0,Y 601.376,Z 270.569,A -85,B 0,C 180,E1 -564.88,E2 -564.88} C_VEL
LIN {X 0,Y 601.389,Z 270.572,A -85,B 0,C 180,E1 -567.36,E2 -567.36} C_VEL
LIN {X 0,Y 601.42,Z 270.567,A -85,B 0,C 180,E1 -570.165,E2 -570.165} C_VEL
LIN {X 0,Y 601.394,Z 270.567,A -85,B 0,C 180,E1 -572.713,E2 -572.713} C_VEL
LIN {X 0,Y 601.375,Z 270.573,A -85,B 0,C 180,E1 -575.111,E2 -575.111} C_VEL
LIN {X 0,Y 601.425,Z 270.573,A -85,B 0,C 180,E1 -577.42,E2 -577.42} C_VEL
LIN {X 0,Y 601.397,Z 270.569,A -85,B 0,C 180,E1 -579.996,E2 -579.996} C_VEL
LIN {X 0,Y 601.372,Z 270.571,A -85,B 0,C 180,E1 -582.674,E2 -582.674} C_VEL
LIN {X 0,Y 601.422,Z 270.571,A -85,B 0,C 180,E1 -585.483,E2 -585.483} C_VEL
LIN {X 0,Y 601.408,Z 270.566,A -85,B 0,C 180,E1 -588.409,E2 -588.409} C_VEL
LIN {X 0,Y 601.427,Z 270.567,A -85,B 0,C 180,E1 -591.53,E2 -591.53} C_VEL
LIN {X 0,Y 601.377,Z 270.57,A -85,B 0,C 180,E1 -594.246,E2 -594.246} C_VEL
LIN {X 0,Y 601.412,Z 270.57,A -85,B 0,C 180,E1 -596.687,E2 -596.687} C_VEL
LIN {X 0,Y 601.402,Z 270.574,A -85,B 0,C 180,E1 -599.058,E2 -599.058} C_VEL
LIN {X 0,Y 601.433,Z 270.565,A -85,B 0,C 180,E1 -601.374,E2 -601.374} C_VEL
LIN {X 0,Y 601.397,Z 270.567,A -85,B 0,C 180,E1 -603.637,E2 -603.637} C_VEL
LIN {X 0,Y 601.411,Z 270.573,A -85,B 0,C 180,E1 -606.59,E2 -606.59} C_VEL
LIN {X 0,Y 601.426,Z 270.563,A -85,B 0,C 180,E1 -609.479,E2 -609.479} C_VEL
LIN {X 0,Y 601.43,Z 270.677,A -85,B 0,C 180,E1 -611.918,E2 -611.918} C_VEL
LIN {X 0,Y 601.459,Z 284.613,A -85,B 0,C 180,E1 -614.411,E2 -614.411} C_VEL
LIN {X 0,Y 601.434,Z 298.826,A -85,B 0,C 180,E1 -616.894,E2 -616.894} C_VEL
LIN {X 0,Y 601.676,Z 305.978,A -85,B 0,C 180,E1 -616.985,E2 -616.985} C_VEL
LIN {X 0,Y 601.624,Z 404.85,A -85,B 0,C 180,E1 -618.183,E2 -618.183} C_VEL
LIN {X 0,Y 601.561,Z 417.419,A -85,B 0,C 180,E1 -618.46,E2 -618.46} C_VEL
LIN {X 0,Y 601.54,Z 430.542,A -85,B 0,C 180,E1 -618.894,E2 -618.894} C_VEL
LIN {X 0,Y 601.525,Z 441.764,A -85,B 0,C 180,E1 -619.397,E2 -619.397} C_VEL
LIN {X 0,Y 601.487,Z 453.538,A -85,B 0,C 180,E1 -620.077,E2 -620.077} C_VEL
LIN {X 0,Y 601.444,Z 464.045,A -85,B 0,C 180,E1 -620.84,E2 -620.84} C_VEL
LIN {X 0,Y 601.429,Z 472.652,A -85,B 0,C 180,E1 -621.602,E2 -621.602} C_VEL
LIN {X 0,Y 601.417,Z 480.577,A -85,B 0,C 180,E1 -622.447,E2 -622.447} C_VEL
LIN {X 0,Y 601.376,Z 487.892,A -85,B 0,C 180,E1 -623.394,E2 -623.394} C_VEL
LIN {X 0,Y 601.372,Z 493.614,A -85,B 0,C 180,E1 -624.3,E2 -624.3} C_VEL
LIN {X 0,Y 601.335,Z 498.757,A -85,B 0,C 180,E1 -625.308,E2 -625.308} C_VEL
LIN {X 0,Y 601.367,Z 502.745,A -85,B 0,C 180,E1 -626.315,E2 -626.315} C_VEL
LIN {X 0,Y 601.324,Z 505.693,A -85,B 0,C 180,E1 -627.321,E2 -627.321} C_VEL
LIN {X 0,Y 601.343,Z 507.128,A -85,B 0,C 180,E1 -627.991,E2 -627.991} C_VEL
LIN {X 0,Y 601.339,Z 508.753,A -85,B 0,C 180,E1 -629.331,E2 -629.331} C_VEL
LIN {X 0,Y 601.336,Z 508.996,A -85,B 0,C 180,E1 -630.001,E2 -630.001} C_VEL
LIN {X 0,Y 601.339,Z 508.814,A -85,B 0,C 180,E1 -630.67,E2 -630.67} C_VEL
LIN {X 0,Y 601.343,Z 507.274,A -85,B 0,C 180,E1 -632.01,E2 -632.01} C_VEL
LIN {X 0,Y 601.326,Z 505.916,A -85,B 0,C 180,E1 -632.68,E2 -632.68} C_VEL
LIN {X 0,Y 601.368,Z 503.039,A -85,B 0,C 180,E1 -633.686,E2 -633.686} C_VEL
LIN {X 0,Y 601.337,Z 499.14,A -85,B 0,C 180,E1 -634.693,E2 -634.693} C_VEL
LIN {X 0,Y 601.373,Z 494.109,A -85,B 0,C 180,E1 -635.702,E2 -635.702} C_VEL
LIN {X 0,Y 601.383,Z 487.785,A -85,B 0,C 180,E1 -636.712,E2 -636.712} C_VEL
LIN {X 0,Y 601.396,Z 479.872,A -85,B 0,C 180,E1 -637.724,E2 -637.724} C_VEL
LIN {X 0,Y 601.437,Z 470.022,A -85,B 0,C 180,E1 -638.738,E2 -638.738} C_VEL
LIN {X 0,Y 601.451,Z 459.702,A -85,B 0,C 180,E1 -639.586,E2 -639.586} C_VEL
LIN {X 0,Y 601.483,Z 448.088,A -85,B 0,C 180,E1 -640.35,E2 -640.35} C_VEL
LIN {X 0,Y 601.526,Z 436.198,A -85,B 0,C 180,E1 -640.959,E2 -640.959} C_VEL
LIN {X 0,Y 601.541,Z 423.239,A -85,B 0,C 180,E1 -641.457,E2 -641.457} C_VEL
LIN {X 0,Y 601.609,Z 410.594,A -85,B 0,C 180,E1 -641.797,E2 -641.797} C_VEL
LIN {X 0,Y 601.616,Z 397.445,A -85,B 0,C 180,E1 -642.011,E2 -642.011} C_VEL
LIN {X 0,Y 601.567,Z 299.72,A -85,B 0,C 180,E1 -643.182,E2 -643.182} C_VEL
LIN {X 0,Y 601.407,Z 298.565,A -85,B 0,C 180,E1 -643.216,E2 -643.216} C_VEL
LIN {X 0,Y 601.431,Z 283.155,A -85,B 0,C 180,E1 -645.939,E2 -645.939} C_VEL
LIN {X 0,Y 601.4,Z 270.569,A -85,B 0,C 180,E1 -648.217,E2 -648.217} C_VEL
LIN {X 0,Y 601.438,Z 270.563,A -85,B 0,C 180,E1 -650.799,E2 -650.799} C_VEL
LIN {X 0,Y 601.415,Z 270.575,A -85,B 0,C 180,E1 -653.411,E2 -653.411} C_VEL
LIN {X 0,Y 601.399,Z 270.566,A -85,B 0,C 180,E1 -656.364,E2 -656.364} C_VEL
LIN {X 0,Y 601.441,Z 270.563,A -85,B 0,C 180,E1 -658.789,E2 -658.789} C_VEL
LIN {X 0,Y 601.402,Z 270.569,A -85,B 0,C 180,E1 -661.727,E2 -661.727} C_VEL
LIN {X 0,Y 601.422,Z 270.564,A -85,B 0,C 180,E1 -664.119,E2 -664.119} C_VEL
LIN {X 0,Y 601.44,Z 270.568,A -85,B 0,C 180,E1 -667.382,E2 -667.382} C_VEL
LIN {X 0,Y 601.404,Z 270.566,A -85,B 0,C 180,E1 -669.996,E2 -669.996} C_VEL
LIN {X 0,Y 601.417,Z 270.568,A -85,B 0,C 180,E1 -672.67,E2 -672.67} C_VEL
LIN {X 0,Y 601.403,Z 270.569,A -85,B 0,C 180,E1 -675.48,E2 -675.48} C_VEL
LIN {X 0,Y 601.425,Z 270.565,A -85,B 0,C 180,E1 -678.407,E2 -678.407} C_VEL
LIN {X 0,Y 601.434,Z 270.571,A -85,B 0,C 180,E1 -680.875,E2 -680.875} C_VEL
LIN {X 0,Y 601.404,Z 270.568,A -85,B 0,C 180,E1 -683.417,E2 -683.417} C_VEL
LIN {X 0,Y 601.435,Z 270.562,A -85,B 0,C 180,E1 -686.065,E2 -686.065} C_VEL
LIN {X 0,Y 601.415,Z 270.57,A -85,B 0,C 180,E1 -689.058,E2 -689.058} C_VEL
LIN {X 0,Y 601.418,Z 270.565,A -85,B 0,C 180,E1 -691.372,E2 -691.372} C_VEL
LIN {X 0,Y 601.397,Z 270.566,A -85,B 0,C 180,E1 -693.636,E2 -693.636} C_VEL
LIN {X 0,Y 601.418,Z 270.573,A -85,B 0,C 180,E1 -696.589,E2 -696.589} C_VEL
LIN {X 0,Y 601.423,Z 270.564,A -85,B 0,C 180,E1 -699.478,E2 -699.478} C_VEL
LIN {X 0,Y 601.453,Z 270.672,A -85,B 0,C 180,E1 -701.918,E2 -701.918} C_VEL
LIN {X 0,Y 601.419,Z 284.608,A -85,B 0,C 180,E1 -704.409,E2 -704.409} C_VEL
LIN {X 0,Y 601.42,Z 298.754,A -85,B 0,C 180,E1 -706.893,E2 -706.893} C_VEL
LIN {X 0,Y 601.659,Z 309.483,A -85,B 0,C 180,E1 -707.027,E2 -707.027} C_VEL
LIN {X 0,Y 601.591,Z 404.766,A -85,B 0,C 180,E1 -708.182,E2 -708.182} C_VEL
LIN {X 0,Y 601.586,Z 418.151,A -85,B 0,C 180,E1 -708.481,E2 -708.481} C_VEL
LIN {X 0,Y 601.574,Z 429.499,A -85,B 0,C 180,E1 -708.855,E2 -708.855} C_VEL
LIN {X 0,Y 601.521,Z 441.721,A -85,B 0,C 180,E1 -709.396,E2 -709.396} C_VEL
LIN {X 0,Y 601.471,Z 453.526,A -85,B 0,C 180,E1 -710.075,E2 -710.075} C_VEL
LIN {X 0,Y 601.438,Z 465.091,A -85,B 0,C 180,E1 -710.924,E2 -710.924} C_VEL
LIN {X 0,Y 601.411,Z 474.349,A -85,B 0,C 180,E1 -711.77,E2 -711.77} C_VEL
LIN {X 0,Y 601.389,Z 483.327,A -85,B 0,C 180,E1 -712.783,E2 -712.783} C_VEL
LIN {X 0,Y 601.376,Z 490.471,A -85,B 0,C 180,E1 -713.781,E2 -713.781} C_VEL
LIN {X 0,Y 601.373,Z 495.44,A -85,B 0,C 180,E1 -714.635,E2 -714.635} C_VEL
LIN {X 0,Y 601.353,Z 500.184,A -85,B 0,C 180,E1 -715.643,E2 -715.643} C_VEL
LIN {X 0,Y 601.345,Z 503.817,A -85,B 0,C 180,E1 -716.65,E2 -716.65} C_VEL
LIN {X 0,Y 601.324,Z 505.688,A -85,B 0,C 180,E1 -717.32,E2 -717.32} C_VEL
LIN {X 0,Y 601.341,Z 507.121,A -85,B 0,C 180,E1 -717.991,E2 -717.991} C_VEL
LIN {X 0,Y 601.349,Z 508.133,A -85,B 0,C 180,E1 -718.661,E2 -718.661} C_VEL
LIN {X 0,Y 601.335,Z 508.989,A -85,B 0,C 180,E1 -720,E2 -720} C_VEL
LIN {X 0,Y 601.339,Z 508.814,A -85,B 0,C 180,E1 -720.67,E2 -720.67} C_VEL
LIN {X 0,Y 601.34,Z 507.273,A -85,B 0,C 180,E1 -722.009,E2 -722.009} C_VEL
LIN {X 0,Y 601.326,Z 505.917,A -85,B 0,C 180,E1 -722.68,E2 -722.68} C_VEL
LIN {X 0,Y 601.368,Z 503.044,A -85,B 0,C 180,E1 -723.685,E2 -723.685} C_VEL
LIN {X 0,Y 601.337,Z 499.144,A -85,B 0,C 180,E1 -724.693,E2 -724.693} C_VEL
LIN {X 0,Y 601.373,Z 494.112,A -85,B 0,C 180,E1 -725.701,E2 -725.701} C_VEL
LIN {X 0,Y 601.383,Z 487.776,A -85,B 0,C 180,E1 -726.711,E2 -726.711} C_VEL
LIN {X 0,Y 601.396,Z 479.876,A -85,B 0,C 180,E1 -727.723,E2 -727.723} C_VEL
LIN {X 0,Y 601.437,Z 470.031,A -85,B 0,C 180,E1 -728.738,E2 -728.738} C_VEL
LIN {X 0,Y 601.446,Z 459.697,A -85,B 0,C 180,E1 -729.585,E2 -729.585} C_VEL
LIN {X 0,Y 601.476,Z 449.483,A -85,B 0,C 180,E1 -730.264,E2 -730.264} C_VEL
LIN {X 0,Y 601.541,Z 437.557,A -85,B 0,C 180,E1 -730.897,E2 -730.897} C_VEL
LIN {X 0,Y 601.572,Z 425.569,A -85,B 0,C 180,E1 -731.379,E2 -731.379} C_VEL
LIN {X 0,Y 601.584,Z 412.416,A -85,B 0,C 180,E1 -731.754,E2 -731.754} C_VEL
LIN {X 0,Y 601.594,Z 399.248,A -85,B 0,C 180,E1 -731.989,E2 -731.989} C_VEL
LIN {X 0,Y 601.573,Z 299.656,A -85,B 0,C 180,E1 -733.183,E2 -733.183} C_VEL
LIN {X 0,Y 601.42,Z 298.568,A -85,B 0,C 180,E1 -733.215,E2 -733.215} C_VEL
LIN {X 0,Y 601.448,Z 283.158,A -85,B 0,C 180,E1 -735.938,E2 -735.938} C_VEL
LIN {X 0,Y 601.384,Z 270.571,A -85,B 0,C 180,E1 -738.195,E2 -738.195} C_VEL
LIN {X 0,Y 601.41,Z 270.567,A -85,B 0,C 180,E1 -740.792,E2 -740.792} C_VEL
LIN {X 0,Y 601.374,Z 270.578,A -85,B 0,C 180,E1 -743.412,E2 -743.412} C_VEL
LIN {X 0,Y 601.365,Z 270.572,A -85,B 0,C 180,E1 -745.857,E2 -745.857} C_VEL
LIN {X 0,Y 601.354,Z 270.573,A -85,B 0,C 180,E1 -747.871,E2 -747.871} C_VEL
LIN {X 0,Y 601.371,Z 270.57,A -85,B 0,C 180,E1 -750.167,E2 -750.167} C_VEL
LIN {X 0,Y 601.388,Z 270.574,A -85,B 0,C 180,E1 -752.71,E2 -752.71} C_VEL
LIN {X 0,Y 601.378,Z 270.576,A -85,B 0,C 180,E1 -755.109,E2 -755.109} C_VEL
LIN {X 0,Y 601.385,Z 270.57,A -85,B 0,C 180,E1 -757.423,E2 -757.423} C_VEL
LIN {X 0,Y 601.373,Z 270.571,A -85,B 0,C 180,E1 -759.998,E2 -759.998} C_VEL
LIN {X 0,Y 601.376,Z 270.579,A -85,B 0,C 180,E1 -762.674,E2 -762.674} C_VEL
LIN {X 0,Y 601.368,Z 270.57,A -85,B 0,C 180,E1 -765.476,E2 -765.476} C_VEL
LIN {X 0,Y 601.416,Z 270.574,A -85,B 0,C 180,E1 -768.408,E2 -768.408} C_VEL
LIN {X 0,Y 601.393,Z 270.57,A -85,B 0,C 180,E1 -770.871,E2 -770.871} C_VEL
LIN {X 0,Y 601.384,Z 270.569,A -85,B 0,C 180,E1 -773.415,E2 -773.415} C_VEL
LIN {X 0,Y 601.431,Z 270.571,A -85,B 0,C 180,E1 -776.065,E2 -776.065} C_VEL
LIN {X 0,Y 601.398,Z 270.567,A -85,B 0,C 180,E1 -779.056,E2 -779.056} C_VEL
LIN {X 0,Y 601.407,Z 270.568,A -85,B 0,C 180,E1 -781.371,E2 -781.371} C_VEL
LIN {X 0,Y 601.414,Z 270.571,A -85,B 0,C 180,E1 -784.133,E2 -784.133} C_VEL
LIN {X 0,Y 601.415,Z 270.647,A -85,B 0,C 180,E1 -786.748,E2 -786.748} C_VEL
LIN {X 0,Y 601.69,Z 275.715,A -85,B 0,C 180,E1 -787.452,E2 -787.452} C_VEL
LIN {X 0,Y 601.595,Z 294.746,A -85,B 0,C 180,E1 -790.019,E2 -790.019} C_VEL
LIN {X 0,Y 601.542,Z 314.69,A -85,B 0,C 180,E1 -792.666,E2 -792.666} C_VEL
LIN {X 0,Y 601.486,Z 334.634,A -85,B 0,C 180,E1 -795.277,E2 -795.277} C_VEL
LIN {X 0,Y 601.471,Z 346.434,A -85,B 0,C 180,E1 -796.807,E2 -796.807} C_VEL
LIN {X 0,Y 601.679,Z 354.246,A -85,B 0,C 180,E1 -796.919,E2 -796.919} C_VEL
LIN {X 0,Y 601.613,Z 454.913,A -85,B 0,C 180,E1 -798.139,E2 -798.139} C_VEL
LIN {X 0,Y 601.558,Z 468.193,A -85,B 0,C 180,E1 -798.437,E2 -798.437} C_VEL
LIN {X 0,Y 601.544,Z 480.612,A -85,B 0,C 180,E1 -798.852,E2 -798.852} C_VEL
LIN {X 0,Y 601.525,Z 492.622,A -85,B 0,C 180,E1 -799.396,E2 -799.396} C_VEL
LIN {X 0,Y 601.487,Z 504.189,A -85,B 0,C 180,E1 -800.075,E2 -800.075} C_VEL
LIN {X 0,Y 601.444,Z 514.587,A -85,B 0,C 180,E1 -800.838,E2 -800.838} C_VEL
LIN {X 0,Y 601.429,Z 523.105,A -85,B 0,C 180,E1 -801.6,E2 -801.6} C_VEL
LIN {X 0,Y 601.418,Z 530.955,A -85,B 0,C 180,E1 -802.445,E2 -802.445} C_VEL
LIN {X 0,Y 601.37,Z 538.222,A -85,B 0,C 180,E1 -803.398,E2 -803.398} C_VEL
LIN {X 0,Y 601.372,Z 543.863,A -85,B 0,C 180,E1 -804.298,E2 -804.298} C_VEL
LIN {X 0,Y 601.336,Z 548.947,A -85,B 0,C 180,E1 -805.307,E2 -805.307} C_VEL
LIN {X 0,Y 601.367,Z 552.894,A -85,B 0,C 180,E1 -806.314,E2 -806.314} C_VEL
LIN {X 0,Y 601.325,Z 555.808,A -85,B 0,C 180,E1 -807.32,E2 -807.32} C_VEL
LIN {X 0,Y 601.343,Z 557.201,A -85,B 0,C 180,E1 -807.99,E2 -807.99} C_VEL
LIN {X 0,Y 601.339,Z 558.783,A -85,B 0,C 180,E1 -809.33,E2 -809.33} C_VEL
LIN {X 0,Y 601.335,Z 559,A -85,B 0,C 180,E1 -809.999,E2 -809.999} C_VEL
LIN {X 0,Y 601.348,Z 558.185,A -85,B 0,C 180,E1 -811.339,E2 -811.339} C_VEL
LIN {X 0,Y 601.343,Z 557.203,A -85,B 0,C 180,E1 -812.009,E2 -812.009} C_VEL
LIN {X 0,Y 601.325,Z 555.811,A -85,B 0,C 180,E1 -812.679,E2 -812.679} C_VEL
LIN {X 0,Y 601.367,Z 552.898,A -85,B 0,C 180,E1 -813.685,E2 -813.685} C_VEL
LIN {X 0,Y 601.336,Z 548.953,A -85,B 0,C 180,E1 -814.692,E2 -814.692} C_VEL
LIN {X 0,Y 601.372,Z 542.881,A -85,B 0,C 180,E1 -815.868,E2 -815.868} C_VEL
LIN {X 0,Y 601.381,Z 536.241,A -85,B 0,C 180,E1 -816.879,E2 -816.879} C_VEL
LIN {X 0,Y 601.4,Z 527.996,A -85,B 0,C 180,E1 -817.892,E2 -817.892} C_VEL
LIN {X 0,Y 601.436,Z 519.545,A -85,B 0,C 180,E1 -818.737,E2 -818.737} C_VEL
LIN {X 0,Y 601.442,Z 509.103,A -85,B 0,C 180,E1 -819.584,E2 -819.584} C_VEL
LIN {X 0,Y 601.471,Z 498.77,A -85,B 0,C 180,E1 -820.264,E2 -820.264} C_VEL
LIN {X 0,Y 601.538,Z 486.59,A -85,B 0,C 180,E1 -820.896,E2 -820.896} C_VEL
LIN {X 0,Y 601.553,Z 474.238,A -85,B 0,C 180,E1 -821.378,E2 -821.378} C_VEL
LIN {X 0,Y 601.58,Z 461.472,A -85,B 0,C 180,E1 -821.732,E2 -821.732} C_VEL
LIN {X 0,Y 601.618,Z 449.141,A -85,B 0,C 180,E1 -821.945,E2 -821.945} C_VEL
LIN {X 0,Y 601.559,Z 347.206,A -85,B 0,C 180,E1 -823.168,E2 -823.168} C_VEL
LIN {X 0,Y 601.463,Z 346.278,A -85,B 0,C 180,E1 -823.213,E2 -823.213} C_VEL
LIN {X 0,Y 601.528,Z 325.337,A -85,B 0,C 180,E1 -825.935,E2 -825.935} C_VEL
LIN {X 0,Y 601.58,Z 303.127,A -85,B 0,C 180,E1 -828.863,E2 -828.863} C_VEL
LIN {X 0,Y 601.685,Z 281.46,A -85,B 0,C 180,E1 -831.768,E2 -831.768} C_VEL
LIN {X 0,Y 601.665,Z 272.153,A -85,B 0,C 180,E1 -833.035,E2 -833.035} C_VEL
LIN {X 0,Y 601.402,Z 270.57,A -85,B 0,C 180,E1 -833.273,E2 -833.273} C_VEL
LIN {X 0,Y 601.414,Z 270.571,A -85,B 0,C 180,E1 -835.867,E2 -835.867} C_VEL
LIN {X 0,Y 601.413,Z 270.566,A -85,B 0,C 180,E1 -838.784,E2 -838.784} C_VEL
LIN {X 0,Y 601.416,Z 270.567,A -85,B 0,C 180,E1 -841.454,E2 -841.454} C_VEL
LIN {X 0,Y 601.421,Z 270.571,A -85,B 0,C 180,E1 -844.118,E2 -844.118} C_VEL
LIN {X 0,Y 601.384,Z 270.569,A -85,B 0,C 180,E1 -846.583,E2 -846.583} C_VEL
LIN {X 0,Y 601.414,Z 270.571,A -85,B 0,C 180,E1 -849.532,E2 -849.532} C_VEL
LIN {X 0,Y 601.412,Z 270.575,A -85,B 0,C 180,E1 -851.765,E2 -851.765} C_VEL
LIN {X 0,Y 601.392,Z 270.567,A -85,B 0,C 180,E1 -854.532,E2 -854.532} C_VEL
LIN {X 0,Y 601.407,Z 270.573,A -85,B 0,C 180,E1 -857.408,E2 -857.408} C_VEL
LIN {X 0,Y 601.389,Z 270.57,A -85,B 0,C 180,E1 -860.003,E2 -860.003} C_VEL
LIN {X 0,Y 601.423,Z 270.564,A -85,B 0,C 180,E1 -862.618,E2 -862.618} C_VEL
LIN {X 0,Y 601.405,Z 270.568,A -85,B 0,C 180,E1 -865.88,E2 -865.88} C_VEL
LIN {X 0,Y 601.405,Z 270.566,A -85,B 0,C 180,E1 -868.546,E2 -868.546} C_VEL
LIN {X 0,Y 601.418,Z 270.572,A -85,B 0,C 180,E1 -871.372,E2 -871.372} C_VEL
LIN {X 0,Y 601.378,Z 270.572,A -85,B 0,C 180,E1 -873.635,E2 -873.635} C_VEL
LIN {X 0,Y 601.387,Z 270.569,A -85,B 0,C 180,E1 -875.857,E2 -875.857} C_VEL
LIN {X 0,Y 601.371,Z 270.57,A -85,B 0,C 180,E1 -878.039,E2 -878.039} C_VEL
LIN {X 0,Y 601.374,Z 270.57,A -85,B 0,C 180,E1 -880.189,E2 -880.189} C_VEL
LIN {X 0,Y 601.395,Z 270.576,A -85,B 0,C 180,E1 -883.013,E2 -883.013} C_VEL
LIN {X 0,Y 601.366,Z 270.571,A -85,B 0,C 180,E1 -885.793,E2 -885.793} C_VEL
LIN {X 0,Y 601.42,Z 270.57,A -85,B 0,C 180,E1 -888.542,E2 -888.542} C_VEL
LIN {X 0,Y 601.374,Z 270.572,A -85,B 0,C 180,E1 -891.261,E2 -891.261} C_VEL
LIN {X 0,Y 601.372,Z 270.571,A -85,B 0,C 180,E1 -893.385,E2 -893.385} C_VEL
LIN {X 0,Y 601.365,Z 270.572,A -85,B 0,C 180,E1 -895.308,E2 -895.308} C_VEL
LIN {X 0,Y 601.385,Z 270.569,A -85,B 0,C 180,E1 -897.321,E2 -897.321} C_VEL
LIN {X 0,Y 601.403,Z 270.569,A -85,B 0,C 180,E1 -900,E2 -900} C_VEL
LIN {X 0,Y 601.425,Z 270.569,A -85,B 0,C 180,E1 -902.679,E2 -902.679} C_VEL
LIN {X 0,Y 601.373,Z 270.57,A -85,B 0,C 180,E1 -905.365,E2 -905.365} C_VEL
LIN {X 0,Y 601.356,Z 270.572,A -85,B 0,C 180,E1 -907.386,E2 -907.386} C_VEL
LIN {X 0,Y 601.406,Z 270.574,A -85,B 0,C 180,E1 -910.096,E2 -910.096} C_VEL
LIN {X 0,Y 601.383,Z 270.574,A -85,B 0,C 180,E1 -912.371,E2 -912.371} C_VEL
LIN {X 0,Y 600.71,Z 270.655,A -85,B 0,C 180,E1 -912.93,E2 -912.93} C_VEL
LIN {X 0,Y 597.852,Z 271.014,A -85,B 0,C 180,E1 -913.838,E2 -913.838} C_VEL
LIN {X 0,Y 595.441,Z 271.312,A -85,B 0,C 180,E1 -914.568,E2 -914.568} C_VEL
LIN {X 0,Y 594.408,Z 271.438,A -85,B 0,C 180,E1 -915.132,E2 -915.132} C_VEL
LIN {X 0,Y 594.324,Z 271.449,A -85,B 0,C 180,E1 -915.323,E2 -915.323} C_VEL
LIN {X 0,Y 594.33,Z 271.456,A -85,B 0,C 180,E1 -917.906,E2 -917.906} C_VEL
LIN {X 0,Y 594.376,Z 271.442,A -85,B 0,C 180,E1 -920.777,E2 -920.777} C_VEL
LIN {X 0,Y 594.367,Z 271.451,A -85,B 0,C 180,E1 -923.705,E2 -923.705} C_VEL
LIN {X 0,Y 594.349,Z 271.445,A -85,B 0,C 180,E1 -926.701,E2 -926.701} C_VEL
LIN {X 0,Y 594.364,Z 271.444,A -85,B 0,C 180,E1 -929,E2 -929} C_VEL
LIN {X 0,Y 594.366,Z 271.453,A -85,B 0,C 180,E1 -931.643,E2 -931.643} C_VEL
LIN {X 0,Y 594.359,Z 271.444,A -85,B 0,C 180,E1 -934.582,E2 -934.582} C_VEL
LIN {X 0,Y 594.379,Z 271.449,A -85,B 0,C 180,E1 -937.609,E2 -937.609} C_VEL
LIN {X 0,Y 594.352,Z 271.445,A -85,B 0,C 180,E1 -940.569,E2 -940.569} C_VEL
LIN {X 0,Y 594.353,Z 271.454,A -85,B 0,C 180,E1 -943.301,E2 -943.301} C_VEL
LIN {X 0,Y 594.346,Z 271.445,A -85,B 0,C 180,E1 -946.163,E2 -946.163} C_VEL
LIN {X 0,Y 594.367,Z 271.444,A -85,B 0,C 180,E1 -948.536,E2 -948.536} C_VEL
LIN {X 0,Y 594.377,Z 271.449,A -85,B 0,C 180,E1 -951.297,E2 -951.297} C_VEL
LIN {X 0,Y 594.347,Z 271.446,A -85,B 0,C 180,E1 -953.756,E2 -953.756} C_VEL
LIN {X 0,Y 594.352,Z 271.445,A -85,B 0,C 180,E1 -956.238,E2 -956.238} C_VEL
LIN {X 0,Y 594.363,Z 271.449,A -85,B 0,C 180,E1 -958.65,E2 -958.65} C_VEL
LIN {X 0,Y 594.382,Z 271.448,A -85,B 0,C 180,E1 -961.043,E2 -961.043} C_VEL
LIN {X 0,Y 594.383,Z 271.444,A -85,B 0,C 180,E1 -963.301,E2 -963.301} C_VEL
LIN {X 0,Y 594.379,Z 271.444,A -85,B 0,C 180,E1 -966.296,E2 -966.296} C_VEL
LIN {X 0,Y 594.404,Z 271.44,A -85,B 0,C 180,E1 -969.225,E2 -969.225} C_VEL
LIN {X 0,Y 594.362,Z 271.536,A -85,B 0,C 180,E1 -971.851,E2 -971.851} C_VEL
LIN {X 0,Y 594.416,Z 284.616,A -85,B 0,C 180,E1 -974.221,E2 -974.221} C_VEL
LIN {X 0,Y 594.364,Z 298.645,A -85,B 0,C 180,E1 -976.73,E2 -976.73} C_VEL
LIN {X 0,Y 594.776,Z 304.235,A -85,B 0,C 180,E1 -976.81,E2 -976.81} C_VEL
LIN {X 0,Y 594.677,Z 404.867,A -85,B 0,C 180,E1 -978.043,E2 -978.043} C_VEL
LIN {X 0,Y 594.619,Z 418.207,A -85,B 0,C 180,E1 -978.345,E2 -978.345} C_VEL
LIN {X 0,Y 594.559,Z 431.31,A -85,B 0,C 180,E1 -978.792,E2 -978.792} C_VEL
LIN {X 0,Y 594.518,Z 443.417,A -85,B 0,C 180,E1 -979.357,E2 -979.357} C_VEL
LIN {X 0,Y 594.475,Z 454.827,A -85,B 0,C 180,E1 -980.044,E2 -980.044} C_VEL
LIN {X 0,Y 594.406,Z 465.106,A -85,B 0,C 180,E1 -980.816,E2 -980.816} C_VEL
LIN {X 0,Y 594.372,Z 474.375,A -85,B 0,C 180,E1 -981.672,E2 -981.672} C_VEL
LIN {X 0,Y 594.316,Z 483.344,A -85,B 0,C 180,E1 -982.697,E2 -982.697} C_VEL
LIN {X 0,Y 594.285,Z 489.86,A -85,B 0,C 180,E1 -983.612,E2 -983.612} C_VEL
LIN {X 0,Y 594.289,Z 495.448,A -85,B 0,C 180,E1 -984.572,E2 -984.572} C_VEL
LIN {X 0,Y 594.27,Z 500.189,A -85,B 0,C 180,E1 -985.592,E2 -985.592} C_VEL
LIN {X 0,Y 594.267,Z 503.82,A -85,B 0,C 180,E1 -986.611,E2 -986.611} C_VEL
LIN {X 0,Y 594.225,Z 505.694,A -85,B 0,C 180,E1 -987.289,E2 -987.289} C_VEL
LIN {X 0,Y 594.242,Z 507.128,A -85,B 0,C 180,E1 -987.967,E2 -987.967} C_VEL
LIN {X 0,Y 594.24,Z 508.753,A -85,B 0,C 180,E1 -989.323,E2 -989.323} C_VEL
LIN {X 0,Y 594.236,Z 508.996,A -85,B 0,C 180,E1 -990.001,E2 -990.001} C_VEL
LIN {X 0,Y 594.239,Z 508.814,A -85,B 0,C 180,E1 -990.678,E2 -990.678} C_VEL
LIN {X 0,Y 594.242,Z 507.272,A -85,B 0,C 180,E1 -992.034,E2 -992.034} C_VEL
LIN {X 0,Y 594.226,Z 505.914,A -85,B 0,C 180,E1 -992.712,E2 -992.712} C_VEL
LIN {X 0,Y 594.289,Z 503.039,A -85,B 0,C 180,E1 -993.73,E2 -993.73} C_VEL
LIN {X 0,Y 594.242,Z 499.139,A -85,B 0,C 180,E1 -994.749,E2 -994.749} C_VEL
LIN {X 0,Y 594.3,Z 494.108,A -85,B 0,C 180,E1 -995.77,E2 -995.77} C_VEL
LIN {X 0,Y 594.317,Z 487.779,A -85,B 0,C 180,E1 -996.792,E2 -996.792} C_VEL
LIN {X 0,Y 594.347,Z 479.87,A -85,B 0,C 180,E1 -997.816,E2 -997.816} C_VEL
LIN {X 0,Y 594.381,Z 470.014,A -85,B 0,C 180,E1 -998.843,E2 -998.843} C_VEL
LIN {X 0,Y 594.435,Z 459.698,A -85,B 0,C 180,E1 -999.7,E2 -999.7} C_VEL
LIN {X 0,Y 594.492,Z 448.082,A -85,B 0,C 180,E1 -1000.473,E2 -1000.473} C_VEL
LIN {X 0,Y 594.55,Z 436.159,A -85,B 0,C 180,E1 -1001.09,E2 -1001.09} C_VEL
LIN {X 0,Y 594.578,Z 423.23,A -85,B 0,C 180,E1 -1001.593,E2 -1001.593} C_VEL
LIN {X 0,Y 594.663,Z 410.556,A -85,B 0,C 180,E1 -1001.937,E2 -1001.937} C_VEL
LIN {X 0,Y 594.698,Z 397.4,A -85,B 0,C 180,E1 -1002.152,E2 -1002.152} C_VEL
LIN {X 0,Y 594.61,Z 300.234,A -85,B 0,C 180,E1 -1003.333,E2 -1003.333} C_VEL
LIN {X 0,Y 594.386,Z 298.562,A -85,B 0,C 180,E1 -1003.375,E2 -1003.375} C_VEL
LIN {X 0,Y 594.405,Z 283.152,A -85,B 0,C 180,E1 -1006.133,E2 -1006.133} C_VEL
LIN {X 0,Y 594.379,Z 271.444,A -85,B 0,C 180,E1 -1008.261,E2 -1008.261} C_VEL
LIN {X 0,Y 594.383,Z 271.443,A -85,B 0,C 180,E1 -1010.916,E2 -1010.916} C_VEL
LIN {X 0,Y 594.383,Z 271.446,A -85,B 0,C 180,E1 -1013.705,E2 -1013.705} C_VEL
LIN {X 0,Y 594.384,Z 271.442,A -85,B 0,C 180,E1 -1016.7,E2 -1016.7} C_VEL
LIN {X 0,Y 594.385,Z 271.445,A -85,B 0,C 180,E1 -1018.999,E2 -1018.999} C_VEL
LIN {X 0,Y 594.38,Z 271.445,A -85,B 0,C 180,E1 -1021.642,E2 -1021.642} C_VEL
LIN {X 0,Y 594.379,Z 271.442,A -85,B 0,C 180,E1 -1024.581,E2 -1024.581} C_VEL
LIN {X 0,Y 594.392,Z 271.443,A -85,B 0,C 180,E1 -1027.608,E2 -1027.608} C_VEL
LIN {X 0,Y 594.369,Z 271.444,A -85,B 0,C 180,E1 -1030.568,E2 -1030.568} C_VEL
LIN {X 0,Y 594.371,Z 271.448,A -85,B 0,C 180,E1 -1033.3,E2 -1033.3} C_VEL
LIN {X 0,Y 594.364,Z 271.443,A -85,B 0,C 180,E1 -1036.162,E2 -1036.162} C_VEL
LIN {X 0,Y 594.382,Z 271.444,A -85,B 0,C 180,E1 -1038.536,E2 -1038.536} C_VEL
LIN {X 0,Y 594.382,Z 271.445,A -85,B 0,C 180,E1 -1041.297,E2 -1041.297} C_VEL
LIN {X 0,Y 594.355,Z 271.444,A -85,B 0,C 180,E1 -1043.756,E2 -1043.756} C_VEL
LIN {X 0,Y 594.379,Z 271.442,A -85,B 0,C 180,E1 -1046.239,E2 -1046.239} C_VEL
LIN {X 0,Y 594.373,Z 271.449,A -85,B 0,C 180,E1 -1048.65,E2 -1048.65} C_VEL
LIN {X 0,Y 594.381,Z 271.446,A -85,B 0,C 180,E1 -1051.043,E2 -1051.043} C_VEL
LIN {X 0,Y 594.382,Z 271.442,A -85,B 0,C 180,E1 -1053.3,E2 -1053.3} C_VEL
LIN {X 0,Y 594.391,Z 271.443,A -85,B 0,C 180,E1 -1056.296,E2 -1056.296} C_VEL
LIN {X 0,Y 594.397,Z 271.441,A -85,B 0,C 180,E1 -1059.224,E2 -1059.224} C_VEL
LIN {X 0,Y 594.385,Z 271.531,A -85,B 0,C 180,E1 -1061.851,E2 -1061.851} C_VEL
LIN {X 0,Y 594.387,Z 284.611,A -85,B 0,C 180,E1 -1064.22,E2 -1064.22} C_VEL
LIN {X 0,Y 594.363,Z 298.8,A -85,B 0,C 180,E1 -1066.734,E2 -1066.734} C_VEL
LIN {X 0,Y 594.749,Z 304.163,A -85,B 0,C 180,E1 -1066.808,E2 -1066.808} C_VEL
LIN {X 0,Y 594.643,Z 404.749,A -85,B 0,C 180,E1 -1068.042,E2 -1068.042} C_VEL
LIN {X 0,Y 594.625,Z 418.181,A -85,B 0,C 180,E1 -1068.344,E2 -1068.344} C_VEL
LIN {X 0,Y 594.591,Z 430.215,A -85,B 0,C 180,E1 -1068.75,E2 -1068.75} C_VEL
LIN {X 0,Y 594.53,Z 441.717,A -85,B 0,C 180,E1 -1069.27,E2 -1069.27} C_VEL
LIN {X 0,Y 594.465,Z 453.539,A -85,B 0,C 180,E1 -1069.957,E2 -1069.957} C_VEL
LIN {X 0,Y 594.406,Z 465.089,A -85,B 0,C 180,E1 -1070.815,E2 -1070.815} C_VEL
LIN {X 0,Y 594.373,Z 474.341,A -85,B 0,C 180,E1 -1071.672,E2 -1071.672} C_VEL
LIN {X 0,Y 594.317,Z 483.332,A -85,B 0,C 180,E1 -1072.697,E2 -1072.697} C_VEL
LIN {X 0,Y 594.285,Z 489.86,A -85,B 0,C 180,E1 -1073.612,E2 -1073.612} C_VEL
LIN {X 0,Y 594.289,Z 495.446,A -85,B 0,C 180,E1 -1074.571,E2 -1074.571} C_VEL
LIN {X 0,Y 594.27,Z 500.189,A -85,B 0,C 180,E1 -1075.591,E2 -1075.591} C_VEL
LIN {X 0,Y 594.268,Z 503.822,A -85,B 0,C 180,E1 -1076.61,E2 -1076.61} C_VEL
LIN {X 0,Y 594.225,Z 505.686,A -85,B 0,C 180,E1 -1077.288,E2 -1077.288} C_VEL
LIN {X 0,Y 594.24,Z 507.113,A -85,B 0,C 180,E1 -1077.967,E2 -1077.967} C_VEL
LIN {X 0,Y 594.248,Z 508.135,A -85,B 0,C 180,E1 -1078.645,E2 -1078.645} C_VEL
LIN {X 0,Y 594.236,Z 508.98,A -85,B 0,C 180,E1 -1080,E2 -1080} C_VEL
LIN {X 0,Y 594.24,Z 508.814,A -85,B 0,C 180,E1 -1080.678,E2 -1080.678} C_VEL
LIN {X 0,Y 594.248,Z 508.238,A -85,B 0,C 180,E1 -1081.355,E2 -1081.355} C_VEL
LIN {X 0,Y 594.226,Z 505.915,A -85,B 0,C 180,E1 -1082.712,E2 -1082.712} C_VEL
LIN {X 0,Y 594.289,Z 503.044,A -85,B 0,C 180,E1 -1083.729,E2 -1083.729} C_VEL
LIN {X 0,Y 594.242,Z 499.144,A -85,B 0,C 180,E1 -1084.749,E2 -1084.749} C_VEL
LIN {X 0,Y 594.299,Z 494.107,A -85,B 0,C 180,E1 -1085.769,E2 -1085.769} C_VEL
LIN {X 0,Y 594.317,Z 487.761,A -85,B 0,C 180,E1 -1086.791,E2 -1086.791} C_VEL
LIN {X 0,Y 594.346,Z 479.872,A -85,B 0,C 180,E1 -1087.816,E2 -1087.816} C_VEL
LIN {X 0,Y 594.382,Z 470.026,A -85,B 0,C 180,E1 -1088.842,E2 -1088.842} C_VEL
LIN {X 0,Y 594.426,Z 459.684,A -85,B 0,C 180,E1 -1089.699,E2 -1089.699} C_VEL
LIN {X 0,Y 594.487,Z 449.464,A -85,B 0,C 180,E1 -1090.386,E2 -1090.386} C_VEL
LIN {X 0,Y 594.557,Z 438.411,A -85,B 0,C 180,E1 -1090.984,E2 -1090.984} C_VEL
LIN {X 0,Y 594.598,Z 425.725,A -85,B 0,C 180,E1 -1091.508,E2 -1091.508} C_VEL
LIN {X 0,Y 594.629,Z 413.288,A -85,B 0,C 180,E1 -1091.872,E2 -1091.872} C_VEL
LIN {X 0,Y 594.685,Z 400.719,A -85,B 0,C 180,E1 -1092.109,E2 -1092.109} C_VEL
LIN {X 0,Y 594.622,Z 300.171,A -85,B 0,C 180,E1 -1093.333,E2 -1093.333} C_VEL
LIN {X 0,Y 594.392,Z 298.565,A -85,B 0,C 180,E1 -1093.374,E2 -1093.374} C_VEL
LIN {X 0,Y 594.408,Z 283.155,A -85,B 0,C 180,E1 -1096.132,E2 -1096.132} C_VEL
LIN {X 0,Y 594.348,Z 271.448,A -85,B 0,C 180,E1 -1098.262,E2 -1098.262} C_VEL
LIN {X 0,Y 594.358,Z 271.447,A -85,B 0,C 180,E1 -1100.91,E2 -1100.91} C_VEL
LIN {X 0,Y 594.339,Z 271.45,A -85,B 0,C 180,E1 -1103.706,E2 -1103.706} C_VEL
LIN {X 0,Y 594.358,Z 271.447,A -85,B 0,C 180,E1 -1106.701,E2 -1106.701} C_VEL
LIN {X 0,Y 594.329,Z 271.449,A -85,B 0,C 180,E1 -1109.779,E2 -1109.779} C_VEL
LIN {X 0,Y 594.336,Z 271.447,A -85,B 0,C 180,E1 -1112.149,E2 -1112.149} C_VEL
LIN {X 0,Y 594.357,Z 271.449,A -85,B 0,C 180,E1 -1114.582,E2 -1114.582} C_VEL
LIN {X 0,Y 594.346,Z 271.446,A -85,B 0,C 180,E1 -1117.602,E2 -1117.602} C_VEL
LIN {X 0,Y 594.356,Z 271.452,A -85,B 0,C 180,E1 -1120.568,E2 -1120.568} C_VEL
LIN {X 0,Y 594.342,Z 271.447,A -85,B 0,C 180,E1 -1123.302,E2 -1123.302} C_VEL
LIN {X 0,Y 594.338,Z 271.451,A -85,B 0,C 180,E1 -1126.164,E2 -1126.164} C_VEL
LIN {X 0,Y 594.36,Z 271.444,A -85,B 0,C 180,E1 -1129.18,E2 -1129.18} C_VEL
LIN {X 0,Y 594.358,Z 271.45,A -85,B 0,C 180,E1 -1132.057,E2 -1132.057} C_VEL
LIN {X 0,Y 594.328,Z 271.451,A -85,B 0,C 180,E1 -1134.68,E2 -1134.68} C_VEL
LIN {X 0,Y 594.376,Z 271.442,A -85,B 0,C 180,E1 -1137.089,E2 -1137.089} C_VEL
LIN {X 0,Y 594.372,Z 271.447,A -85,B 0,C 180,E1 -1139.675,E2 -1139.675} C_VEL
LIN {X 0,Y 594.38,Z 271.444,A -85,B 0,C 180,E1 -1142.539,E2 -1142.539} C_VEL
LIN {X 0,Y 594.403,Z 271.445,A -85,B 0,C 180,E1 -1145.564,E2 -1145.564} C_VEL
LIN {X 0,Y 594.381,Z 271.478,A -85,B 0,C 180,E1 -1146.572,E2 -1146.572} C_VEL
LIN {X 0,Y 594.792,Z 275.655,A -85,B 0,C 180,E1 -1147.168,E2 -1147.168} C_VEL
LIN {X 0,Y 594.679,Z 294.746,A -85,B 0,C 180,E1 -1149.776,E2 -1149.776} C_VEL
LIN {X 0,Y 594.574,Z 314.69,A -85,B 0,C 180,E1 -1152.457,E2 -1152.457} C_VEL
LIN {X 0,Y 594.487,Z 335.963,A -85,B 0,C 180,E1 -1155.275,E2 -1155.275} C_VEL
LIN {X 0,Y 594.449,Z 346.434,A -85,B 0,C 180,E1 -1156.649,E2 -1156.649} C_VEL
LIN {X 0,Y 594.783,Z 350.669,A -85,B 0,C 180,E1 -1156.721,E2 -1156.721} C_VEL
LIN {X 0,Y 594.665,Z 454.913,A -85,B 0,C 180,E1 -1157.998,E2 -1157.998} C_VEL
LIN {X 0,Y 594.6,Z 468.193,A -85,B 0,C 180,E1 -1158.3,E2 -1158.3} C_VEL
LIN {X 0,Y 594.599,Z 480.406,A -85,B 0,C 180,E1 -1158.712,E2 -1158.712} C_VEL
LIN {X 0,Y 594.53,Z 492.621,A -85,B 0,C 180,E1 -1159.269,E2 -1159.269} C_VEL
LIN {X 0,Y 594.481,Z 504.191,A -85,B 0,C 180,E1 -1159.957,E2 -1159.957} C_VEL
LIN {X 0,Y 594.414,Z 514.589,A -85,B 0,C 180,E1 -1160.729,E2 -1160.729} C_VEL
LIN {X 0,Y 594.383,Z 523.106,A -85,B 0,C 180,E1 -1161.5,E2 -1161.5} C_VEL
LIN {X 0,Y 594.347,Z 530.955,A -85,B 0,C 180,E1 -1162.355,E2 -1162.355} C_VEL
LIN {X 0,Y 594.283,Z 538.81,A -85,B 0,C 180,E1 -1163.408,E2 -1163.408} C_VEL
LIN {X 0,Y 594.289,Z 545.677,A -85,B 0,C 180,E1 -1164.571,E2 -1164.571} C_VEL
LIN {X 0,Y 594.27,Z 550.368,A -85,B 0,C 180,E1 -1165.591,E2 -1165.591} C_VEL
LIN {X 0,Y 594.267,Z 553.955,A -85,B 0,C 180,E1 -1166.609,E2 -1166.609} C_VEL
LIN {X 0,Y 594.226,Z 555.808,A -85,B 0,C 180,E1 -1167.288,E2 -1167.288} C_VEL
LIN {X 0,Y 594.242,Z 557.2,A -85,B 0,C 180,E1 -1167.966,E2 -1167.966} C_VEL
LIN {X 0,Y 594.239,Z 558.784,A -85,B 0,C 180,E1 -1169.322,E2 -1169.322} C_VEL
LIN {X 0,Y 594.236,Z 559,A -85,B 0,C 180,E1 -1169.999,E2 -1169.999} C_VEL
LIN {X 0,Y 594.248,Z 558.185,A -85,B 0,C 180,E1 -1171.355,E2 -1171.355} C_VEL
LIN {X 0,Y 594.242,Z 557.202,A -85,B 0,C 180,E1 -1172.033,E2 -1172.033} C_VEL
LIN {X 0,Y 594.226,Z 555.81,A -85,B 0,C 180,E1 -1172.711,E2 -1172.711} C_VEL
LIN {X 0,Y 594.288,Z 552.898,A -85,B 0,C 180,E1 -1173.729,E2 -1173.729} C_VEL
LIN {X 0,Y 594.241,Z 548.953,A -85,B 0,C 180,E1 -1174.748,E2 -1174.748} C_VEL
LIN {X 0,Y 594.304,Z 542.882,A -85,B 0,C 180,E1 -1175.939,E2 -1175.939} C_VEL
LIN {X 0,Y 594.307,Z 536.241,A -85,B 0,C 180,E1 -1176.961,E2 -1176.961} C_VEL
LIN {X 0,Y 594.359,Z 527.996,A -85,B 0,C 180,E1 -1177.986,E2 -1177.986} C_VEL
LIN {X 0,Y 594.382,Z 519.545,A -85,B 0,C 180,E1 -1178.841,E2 -1178.841} C_VEL
LIN {X 0,Y 594.425,Z 509.104,A -85,B 0,C 180,E1 -1179.699,E2 -1179.699} C_VEL
LIN {X 0,Y 594.484,Z 498.771,A -85,B 0,C 180,E1 -1180.386,E2 -1180.386} C_VEL
LIN {X 0,Y 594.56,Z 487.701,A -85,B 0,C 180,E1 -1180.974,E2 -1180.974} C_VEL
LIN {X 0,Y 594.578,Z 475.725,A -85,B 0,C 180,E1 -1181.464,E2 -1181.464} C_VEL
LIN {X 0,Y 594.623,Z 462.386,A -85,B 0,C 180,E1 -1181.85,E2 -1181.85} C_VEL
LIN {X 0,Y 594.695,Z 449.141,A -85,B 0,C 180,E1 -1182.086,E2 -1182.086} C_VEL
LIN {X 0,Y 594.659,Z 347.988,A -85,B 0,C 180,E1 -1183.314,E2 -1183.314} C_VEL
LIN {X 0,Y 594.449,Z 346.445,A -85,B 0,C 180,E1 -1183.35,E2 -1183.35} C_VEL
LIN {X 0,Y 594.529,Z 324.008,A -85,B 0,C 180,E1 -1186.304,E2 -1186.304} C_VEL
LIN {X 0,Y 594.669,Z 301.404,A -85,B 0,C 180,E1 -1189.323,E2 -1189.323} C_VEL
LIN {X 0,Y 594.799,Z 279.023,A -85,B 0,C 180,E1 -1192.368,E2 -1192.368} C_VEL
LIN {X 0,Y 594.748,Z 273.483,A -85,B 0,C 180,E1 -1193.135,E2 -1193.135} C_VEL
LIN {X 0,Y 594.351,Z 271.45,A -85,B 0,C 180,E1 -1193.451,E2 -1193.451} C_VEL
LIN {X 0,Y 594.365,Z 271.452,A -85,B 0,C 180,E1 -1196.018,E2 -1196.018} C_VEL
LIN {X 0,Y 594.374,Z 271.442,A -85,B 0,C 180,E1 -1198.956,E2 -1198.956} C_VEL
LIN {X 0,Y 594.373,Z 271.446,A -85,B 0,C 180,E1 -1201.641,E2 -1201.641} C_VEL
LIN {X 0,Y 594.365,Z 271.444,A -85,B 0,C 180,E1 -1204.58,E2 -1204.58} C_VEL
LIN {X 0,Y 594.382,Z 271.447,A -85,B 0,C 180,E1 -1207.607,E2 -1207.607} C_VEL
LIN {X 0,Y 594.354,Z 271.444,A -85,B 0,C 180,E1 -1210.567,E2 -1210.567} C_VEL
LIN {X 0,Y 594.354,Z 271.448,A -85,B 0,C 180,E1 -1213.299,E2 -1213.299} C_VEL
LIN {X 0,Y 594.336,Z 271.448,A -85,B 0,C 180,E1 -1216.162,E2 -1216.162} C_VEL
LIN {X 0,Y 594.361,Z 271.443,A -85,B 0,C 180,E1 -1218.534,E2 -1218.534} C_VEL
LIN {X 0,Y 594.362,Z 271.45,A -85,B 0,C 180,E1 -1221.297,E2 -1221.297} C_VEL
LIN {X 0,Y 594.339,Z 271.451,A -85,B 0,C 180,E1 -1223.754,E2 -1223.754} C_VEL
LIN {X 0,Y 594.347,Z 271.445,A -85,B 0,C 180,E1 -1226.237,E2 -1226.237} C_VEL
LIN {X 0,Y 594.354,Z 271.446,A -85,B 0,C 180,E1 -1228.649,E2 -1228.649} C_VEL
LIN {X 0,Y 594.372,Z 271.449,A -85,B 0,C 180,E1 -1231.042,E2 -1231.042} C_VEL
LIN {X 0,Y 594.322,Z 271.448,A -85,B 0,C 180,E1 -1233.988,E2 -1233.988} C_VEL
LIN {X 0,Y 594.335,Z 271.447,A -85,B 0,C 180,E1 -1236.294,E2 -1236.294} C_VEL
LIN {X 0,Y 594.379,Z 271.448,A -85,B 0,C 180,E1 -1239.223,E2 -1239.223} C_VEL
LIN {X 0,Y 594.319,Z 271.449,A -85,B 0,C 180,E1 -1242.094,E2 -1242.094} C_VEL
LIN {X 0,Y 594.337,Z 271.448,A -85,B 0,C 180,E1 -1244.218,E2 -1244.218} C_VEL
LIN {X 0,Y 594.323,Z 271.455,A -85,B 0,C 180,E1 -1247.016,E2 -1247.016} C_VEL
LIN {X 0,Y 594.341,Z 271.451,A -85,B 0,C 180,E1 -1249.094,E2 -1249.094} C_VEL
LIN {X 0,Y 594.33,Z 271.448,A -85,B 0,C 180,E1 -1251.842,E2 -1251.842} C_VEL
LIN {X 0,Y 594.372,Z 271.452,A -85,B 0,C 180,E1 -1254.572,E2 -1254.572} C_VEL
LIN {X 0,Y 594.356,Z 271.445,A -85,B 0,C 180,E1 -1257.289,E2 -1257.289} C_VEL
LIN {X 0,Y 594.375,Z 271.445,A -85,B 0,C 180,E1 -1260,E2 -1260} C_VEL
LIN {X 0,Y 594.387,Z 271.445,A -85,B 0,C 180,E1 -1262.711,E2 -1262.711} C_VEL
LIN {X 0,Y 594.341,Z 271.446,A -85,B 0,C 180,E1 -1265.428,E2 -1265.428} C_VEL
LIN {X 0,Y 594.345,Z 271.454,A -85,B 0,C 180,E1 -1268.158,E2 -1268.158} C_VEL
LIN {X 0,Y 594.354,Z 271.444,A -85,B 0,C 180,E1 -1271.061,E2 -1271.061} C_VEL
LIN {X 0,Y 594.353,Z 271.448,A -85,B 0,C 180,E1 -1273.68,E2 -1273.68} C_VEL
LIN {X 0,Y 594.324,Z 271.449,A -85,B 0,C 180,E1 -1275.323,E2 -1275.323} C_VEL
LIN {X 0,Y 593.657,Z 271.539,A -85,B 0,C 180,E1 -1275.888,E2 -1275.888} C_VEL
LIN {X 0,Y 590.797,Z 271.899,A -85,B 0,C 180,E1 -1276.806,E2 -1276.806} C_VEL
LIN {X 0,Y 588.387,Z 272.2,A -85,B 0,C 180,E1 -1277.545,E2 -1277.545} C_VEL
LIN {X 0,Y 587.362,Z 272.324,A -85,B 0,C 180,E1 -1278.115,E2 -1278.115} C_VEL
LIN {X 0,Y 587.284,Z 272.33,A -85,B 0,C 180,E1 -1278.308,E2 -1278.308} C_VEL
LIN {X 0,Y 587.323,Z 272.321,A -85,B 0,C 180,E1 -1281.038,E2 -1281.038} C_VEL
LIN {X 0,Y 587.304,Z 272.324,A -85,B 0,C 180,E1 -1283.26,E2 -1283.26} C_VEL
LIN {X 0,Y 587.316,Z 272.327,A -85,B 0,C 180,E1 -1285.518,E2 -1285.518} C_VEL
LIN {X 0,Y 587.294,Z 272.333,A -85,B 0,C 180,E1 -1287.821,E2 -1287.821} C_VEL
LIN {X 0,Y 587.322,Z 272.321,A -85,B 0,C 180,E1 -1290.509,E2 -1290.509} C_VEL
LIN {X 0,Y 587.326,Z 272.327,A -85,B 0,C 180,E1 -1293.397,E2 -1293.397} C_VEL
LIN {X 0,Y 587.282,Z 272.33,A -85,B 0,C 180,E1 -1295.901,E2 -1295.901} C_VEL
LIN {X 0,Y 587.311,Z 272.322,A -85,B 0,C 180,E1 -1298.481,E2 -1298.481} C_VEL
LIN {X 0,Y 587.328,Z 272.326,A -85,B 0,C 180,E1 -1301.158,E2 -1301.158} C_VEL
LIN {X 0,Y 587.307,Z 272.323,A -85,B 0,C 180,E1 -1304.113,E2 -1304.113} C_VEL
LIN {X 0,Y 587.303,Z 272.329,A -85,B 0,C 180,E1 -1306.994,E2 -1306.994} C_VEL
LIN {X 0,Y 587.305,Z 272.324,A -85,B 0,C 180,E1 -1309.746,E2 -1309.746} C_VEL
LIN {X 0,Y 587.338,Z 272.319,A -85,B 0,C 180,E1 -1312.393,E2 -1312.393} C_VEL
LIN {X 0,Y 587.336,Z 272.32,A -85,B 0,C 180,E1 -1315.654,E2 -1315.654} C_VEL
LIN {X 0,Y 587.337,Z 272.319,A -85,B 0,C 180,E1 -1318.232,E2 -1318.232} C_VEL
LIN {X 0,Y 587.346,Z 272.327,A -85,B 0,C 180,E1 -1320.868,E2 -1320.868} C_VEL
LIN {X 0,Y 587.335,Z 272.319,A -85,B 0,C 180,E1 -1323.722,E2 -1323.722} C_VEL
LIN {X 0,Y 587.321,Z 272.321,A -85,B 0,C 180,E1 -1325.994,E2 -1325.994} C_VEL
LIN {X 0,Y 587.318,Z 272.324,A -85,B 0,C 180,E1 -1328.226,E2 -1328.226} C_VEL
LIN {X 0,Y 587.349,Z 272.321,A -85,B 0,C 180,E1 -1331.152,E2 -1331.152} C_VEL
LIN {X 0,Y 587.33,Z 272.395,A -85,B 0,C 180,E1 -1331.784,E2 -1331.784} C_VEL
LIN {X 0,Y 587.402,Z 282.664,A -85,B 0,C 180,E1 -1333.671,E2 -1333.671} C_VEL
LIN {X 0,Y 587.331,Z 298.556,A -85,B 0,C 180,E1 -1336.551,E2 -1336.551} C_VEL
LIN {X 0,Y 587.873,Z 302.492,A -85,B 0,C 180,E1 -1336.63,E2 -1336.63} C_VEL
LIN {X 0,Y 587.738,Z 404.883,A -85,B 0,C 180,E1 -1337.9,E2 -1337.9} C_VEL
LIN {X 0,Y 587.686,Z 418.236,A -85,B 0,C 180,E1 -1338.205,E2 -1338.205} C_VEL
LIN {X 0,Y 587.594,Z 430.715,A -85,B 0,C 180,E1 -1338.632,E2 -1338.632} C_VEL
LIN {X 0,Y 587.532,Z 443.432,A -85,B 0,C 180,E1 -1339.229,E2 -1339.229} C_VEL
LIN {X 0,Y 587.468,Z 454.839,A -85,B 0,C 180,E1 -1339.924,E2 -1339.924} C_VEL
LIN {X 0,Y 587.383,Z 465.109,A -85,B 0,C 180,E1 -1340.705,E2 -1340.705} C_VEL
LIN {X 0,Y 587.34,Z 474.383,A -85,B 0,C 180,E1 -1341.572,E2 -1341.572} C_VEL
LIN {X 0,Y 587.259,Z 483.351,A -85,B 0,C 180,E1 -1342.609,E2 -1342.609} C_VEL
LIN {X 0,Y 587.198,Z 490.435,A -85,B 0,C 180,E1 -1343.624,E2 -1343.624} C_VEL
LIN {X 0,Y 587.211,Z 495.453,A -85,B 0,C 180,E1 -1344.506,E2 -1344.506} C_VEL
LIN {X 0,Y 587.188,Z 500.193,A -85,B 0,C 180,E1 -1345.539,E2 -1345.539} C_VEL
LIN {X 0,Y 587.193,Z 503.822,A -85,B 0,C 180,E1 -1346.57,E2 -1346.57} C_VEL
LIN {X 0,Y 587.131,Z 505.694,A -85,B 0,C 180,E1 -1347.256,E2 -1347.256} C_VEL
LIN {X 0,Y 587.141,Z 507.129,A -85,B 0,C 180,E1 -1347.943,E2 -1347.943} C_VEL
LIN {X 0,Y 587.14,Z 508.754,A -85,B 0,C 180,E1 -1349.315,E2 -1349.315} C_VEL
LIN {X 0,Y 587.137,Z 508.996,A -85,B 0,C 180,E1 -1350.001,E2 -1350.001} C_VEL
LIN {X 0,Y 587.14,Z 508.814,A -85,B 0,C 180,E1 -1350.687,E2 -1350.687} C_VEL
LIN {X 0,Y 587.141,Z 507.271,A -85,B 0,C 180,E1 -1352.059,E2 -1352.059} C_VEL
LIN {X 0,Y 587.133,Z 505.912,A -85,B 0,C 180,E1 -1352.745,E2 -1352.745} C_VEL
LIN {X 0,Y 587.213,Z 503.038,A -85,B 0,C 180,E1 -1353.775,E2 -1353.775} C_VEL
LIN {X 0,Y 587.147,Z 499.139,A -85,B 0,C 180,E1 -1354.807,E2 -1354.807} C_VEL
LIN {X 0,Y 587.23,Z 494.107,A -85,B 0,C 180,E1 -1355.839,E2 -1355.839} C_VEL
LIN {X 0,Y 587.231,Z 487.772,A -85,B 0,C 180,E1 -1356.874,E2 -1356.874} C_VEL
LIN {X 0,Y 587.288,Z 479.869,A -85,B 0,C 180,E1 -1357.911,E2 -1357.911} C_VEL
LIN {X 0,Y 587.336,Z 471.798,A -85,B 0,C 180,E1 -1358.776,E2 -1358.776} C_VEL
LIN {X 0,Y 587.391,Z 461.96,A -85,B 0,C 180,E1 -1359.644,E2 -1359.644} C_VEL
LIN {X 0,Y 587.473,Z 450.902,A -85,B 0,C 180,E1 -1360.425,E2 -1360.425} C_VEL
LIN {X 0,Y 587.564,Z 438.646,A -85,B 0,C 180,E1 -1361.106,E2 -1361.106} C_VEL
LIN {X 0,Y 587.621,Z 425.679,A -85,B 0,C 180,E1 -1361.648,E2 -1361.648} C_VEL
LIN {X 0,Y 587.695,Z 412.421,A -85,B 0,C 180,E1 -1362.037,E2 -1362.037} C_VEL
LIN {X 0,Y 587.781,Z 399.125,A -85,B 0,C 180,E1 -1362.276,E2 -1362.276} C_VEL
LIN {X 0,Y 587.776,Z 301.419,A -85,B 0,C 180,E1 -1363.476,E2 -1363.476} C_VEL
LIN {X 0,Y 587.354,Z 298.559,A -85,B 0,C 180,E1 -1363.538,E2 -1363.538} C_VEL
LIN {X 0,Y 587.402,Z 283.149,A -85,B 0,C 180,E1 -1366.33,E2 -1366.33} C_VEL
LIN {X 0,Y 587.335,Z 272.322,A -85,B 0,C 180,E1 -1368.33,E2 -1368.33} C_VEL
LIN {X 0,Y 587.337,Z 272.322,A -85,B 0,C 180,E1 -1371.038,E2 -1371.038} C_VEL
LIN {X 0,Y 587.322,Z 272.328,A -85,B 0,C 180,E1 -1373.259,E2 -1373.259} C_VEL
LIN {X 0,Y 587.332,Z 272.327,A -85,B 0,C 180,E1 -1375.517,E2 -1375.517} C_VEL
LIN {X 0,Y 587.345,Z 272.32,A -85,B 0,C 180,E1 -1377.818,E2 -1377.818} C_VEL
LIN {X 0,Y 587.327,Z 272.32,A -85,B 0,C 180,E1 -1380.508,E2 -1380.508} C_VEL
LIN {X 0,Y 587.342,Z 272.326,A -85,B 0,C 180,E1 -1383.112,E2 -1383.112} C_VEL
LIN {X 0,Y 587.294,Z 272.325,A -85,B 0,C 180,E1 -1385.9,E2 -1385.9} C_VEL
LIN {X 0,Y 587.326,Z 272.321,A -85,B 0,C 180,E1 -1388.48,E2 -1388.48} C_VEL
LIN {X 0,Y 587.338,Z 272.328,A -85,B 0,C 180,E1 -1391.157,E2 -1391.157} C_VEL
LIN {X 0,Y 587.332,Z 272.319,A -85,B 0,C 180,E1 -1394.113,E2 -1394.113} C_VEL
LIN {X 0,Y 587.316,Z 272.331,A -85,B 0,C 180,E1 -1396.993,E2 -1396.993} C_VEL
LIN {X 0,Y 587.318,Z 272.321,A -85,B 0,C 180,E1 -1399.746,E2 -1399.746} C_VEL
LIN {X 0,Y 587.348,Z 272.319,A -85,B 0,C 180,E1 -1402.392,E2 -1402.392} C_VEL
LIN {X 0,Y 587.348,Z 272.317,A -85,B 0,C 180,E1 -1405.653,E2 -1405.653} C_VEL
LIN {X 0,Y 587.341,Z 272.319,A -85,B 0,C 180,E1 -1408.231,E2 -1408.231} C_VEL
LIN {X 0,Y 587.349,Z 272.325,A -85,B 0,C 180,E1 -1410.868,E2 -1410.868} C_VEL
LIN {X 0,Y 587.333,Z 272.318,A -85,B 0,C 180,E1 -1413.721,E2 -1413.721} C_VEL
LIN {X 0,Y 587.339,Z 272.319,A -85,B 0,C 180,E1 -1415.994,E2 -1415.994} C_VEL
LIN {X 0,Y 587.321,Z 272.323,A -85,B 0,C 180,E1 -1418.226,E2 -1418.226} C_VEL
LIN {X 0,Y 587.348,Z 272.321,A -85,B 0,C 180,E1 -1421.151,E2 -1421.151} C_VEL
LIN {X 0,Y 587.352,Z 272.39,A -85,B 0,C 180,E1 -1421.784,E2 -1421.784} C_VEL
LIN {X 0,Y 587.361,Z 284.615,A -85,B 0,C 180,E1 -1424.026,E2 -1424.026} C_VEL
LIN {X 0,Y 587.333,Z 298.847,A -85,B 0,C 180,E1 -1426.572,E2 -1426.572} C_VEL
LIN {X 0,Y 587.838,Z 302.42,A -85,B 0,C 180,E1 -1426.628,E2 -1426.628} C_VEL
LIN {X 0,Y 587.7,Z 404.731,A -85,B 0,C 180,E1 -1427.898,E2 -1427.898} C_VEL
LIN {X 0,Y 587.695,Z 418.211,A -85,B 0,C 180,E1 -1428.205,E2 -1428.205} C_VEL
LIN {X 0,Y 587.61,Z 430.773,A -85,B 0,C 180,E1 -1428.637,E2 -1428.637} C_VEL
LIN {X 0,Y 587.548,Z 441.713,A -85,B 0,C 180,E1 -1429.141,E2 -1429.141} C_VEL
LIN {X 0,Y 587.462,Z 453.551,A -85,B 0,C 180,E1 -1429.836,E2 -1429.836} C_VEL
LIN {X 0,Y 587.383,Z 465.082,A -85,B 0,C 180,E1 -1430.704,E2 -1430.704} C_VEL
LIN {X 0,Y 587.341,Z 474.333,A -85,B 0,C 180,E1 -1431.571,E2 -1431.571} C_VEL
LIN {X 0,Y 587.272,Z 481.967,A -85,B 0,C 180,E1 -1432.436,E2 -1432.436} C_VEL
LIN {X 0,Y 587.247,Z 488.831,A -85,B 0,C 180,E1 -1433.376,E2 -1433.376} C_VEL
LIN {X 0,Y 587.212,Z 495.452,A -85,B 0,C 180,E1 -1434.506,E2 -1434.506} C_VEL
LIN {X 0,Y 587.188,Z 500.194,A -85,B 0,C 180,E1 -1435.538,E2 -1435.538} C_VEL
LIN {X 0,Y 587.194,Z 503.826,A -85,B 0,C 180,E1 -1436.569,E2 -1436.569} C_VEL
LIN {X 0,Y 587.131,Z 505.684,A -85,B 0,C 180,E1 -1437.256,E2 -1437.256} C_VEL
LIN {X 0,Y 587.148,Z 508.136,A -85,B 0,C 180,E1 -1438.628,E2 -1438.628} C_VEL
LIN {X 0,Y 587.14,Z 508.752,A -85,B 0,C 180,E1 -1439.314,E2 -1439.314} C_VEL
LIN {X 0,Y 587.14,Z 508.813,A -85,B 0,C 180,E1 -1440.686,E2 -1440.686} C_VEL
LIN {X 0,Y 587.147,Z 508.239,A -85,B 0,C 180,E1 -1441.372,E2 -1441.372} C_VEL
LIN {X 0,Y 587.133,Z 505.912,A -85,B 0,C 180,E1 -1442.744,E2 -1442.744} C_VEL
LIN {X 0,Y 587.213,Z 503.042,A -85,B 0,C 180,E1 -1443.774,E2 -1443.774} C_VEL
LIN {X 0,Y 587.147,Z 499.142,A -85,B 0,C 180,E1 -1444.806,E2 -1444.806} C_VEL
LIN {X 0,Y 587.229,Z 494.097,A -85,B 0,C 180,E1 -1445.839,E2 -1445.839} C_VEL
LIN {X 0,Y 587.229,Z 487.746,A -85,B 0,C 180,E1 -1446.874,E2 -1446.874} C_VEL
LIN {X 0,Y 587.288,Z 479.868,A -85,B 0,C 180,E1 -1447.91,E2 -1447.91} C_VEL
LIN {X 0,Y 587.343,Z 470.02,A -85,B 0,C 180,E1 -1448.949,E2 -1448.949} C_VEL
LIN {X 0,Y 587.411,Z 459.672,A -85,B 0,C 180,E1 -1449.816,E2 -1449.816} C_VEL
LIN {X 0,Y 587.502,Z 449.441,A -85,B 0,C 180,E1 -1450.511,E2 -1450.511} C_VEL
LIN {X 0,Y 587.572,Z 437.865,A -85,B 0,C 180,E1 -1451.142,E2 -1451.142} C_VEL
LIN {X 0,Y 587.64,Z 425.897,A -85,B 0,C 180,E1 -1451.64,E2 -1451.64} C_VEL
LIN {X 0,Y 587.677,Z 413.239,A -85,B 0,C 180,E1 -1452.015,E2 -1452.015} C_VEL
LIN {X 0,Y 587.741,Z 400.681,A -85,B 0,C 180,E1 -1452.254,E2 -1452.254} C_VEL
LIN {X 0,Y 587.694,Z 300.795,A -85,B 0,C 180,E1 -1453.485,E2 -1453.485} C_VEL
LIN {X 0,Y 587.368,Z 298.562,A -85,B 0,C 180,E1 -1453.537,E2 -1453.537} C_VEL
LIN {X 0,Y 587.397,Z 283.152,A -85,B 0,C 180,E1 -1456.33,E2 -1456.33} C_VEL
LIN {X 0,Y 587.315,Z 272.389,A -85,B 0,C 180,E1 -1458.307,E2 -1458.307} C_VEL
LIN {X 0,Y 587.318,Z 272.326,A -85,B 0,C 180,E1 -1461.038,E2 -1461.038} C_VEL
LIN {X 0,Y 587.298,Z 272.333,A -85,B 0,C 180,E1 -1463.26,E2 -1463.26} C_VEL
LIN {X 0,Y 587.297,Z 272.324,A -85,B 0,C 180,E1 -1466.168,E2 -1466.168} C_VEL
LIN {X 0,Y 587.3,Z 272.333,A -85,B 0,C 180,E1 -1469.124,E2 -1469.124} C_VEL
LIN {X 0,Y 587.296,Z 272.324,A -85,B 0,C 180,E1 -1471.827,E2 -1471.827} C_VEL
LIN {X 0,Y 587.312,Z 272.324,A -85,B 0,C 180,E1 -1474.342,E2 -1474.342} C_VEL
LIN {X 0,Y 587.299,Z 272.324,A -85,B 0,C 180,E1 -1477.611,E2 -1477.611} C_VEL
LIN {X 0,Y 587.298,Z 272.326,A -85,B 0,C 180,E1 -1480.256,E2 -1480.256} C_VEL
LIN {X 0,Y 587.289,Z 272.327,A -85,B 0,C 180,E1 -1483.115,E2 -1483.115} C_VEL
LIN {X 0,Y 587.289,Z 272.327,A -85,B 0,C 180,E1 -1486.046,E2 -1486.046} C_VEL
LIN {X 0,Y 587.312,Z 272.324,A -85,B 0,C 180,E1 -1488.928,E2 -1488.928} C_VEL
LIN {X 0,Y 587.307,Z 272.323,A -85,B 0,C 180,E1 -1491.518,E2 -1491.518} C_VEL
LIN {X 0,Y 587.281,Z 272.333,A -85,B 0,C 180,E1 -1494.099,E2 -1494.099} C_VEL
LIN {X 0,Y 587.339,Z 272.32,A -85,B 0,C 180,E1 -1496.889,E2 -1496.889} C_VEL
LIN {X 0,Y 587.324,Z 272.323,A -85,B 0,C 180,E1 -1499.493,E2 -1499.493} C_VEL
LIN {X 0,Y 587.306,Z 272.33,A -85,B 0,C 180,E1 -1502.18,E2 -1502.18} C_VEL
LIN {X 0,Y 587.354,Z 272.319,A -85,B 0,C 180,E1 -1505.241,E2 -1505.241} C_VEL
LIN {X 0,Y 587.37,Z 272.475,A -85,B 0,C 180,E1 -1506.416,E2 -1506.416} C_VEL
LIN {X 0,Y 587.888,Z 276.491,A -85,B 0,C 180,E1 -1507.001,E2 -1507.001} C_VEL
LIN {X 0,Y 587.754,Z 294.746,A -85,B 0,C 180,E1 -1509.527,E2 -1509.527} C_VEL
LIN {X 0,Y 587.604,Z 316.019,A -85,B 0,C 180,E1 -1512.422,E2 -1512.422} C_VEL
LIN {X 0,Y 587.485,Z 337.293,A -85,B 0,C 180,E1 -1515.273,E2 -1515.273} C_VEL
LIN {X 0,Y 587.407,Z 346.434,A -85,B 0,C 180,E1 -1516.486,E2 -1516.486} C_VEL
LIN {X 0,Y 587.889,Z 350.669,A -85,B 0,C 180,E1 -1516.563,E2 -1516.563} C_VEL
LIN {X 0,Y 587.724,Z 454.913,A -85,B 0,C 180,E1 -1517.854,E2 -1517.854} C_VEL
LIN {X 0,Y 587.668,Z 468.192,A -85,B 0,C 180,E1 -1518.16,E2 -1518.16} C_VEL
LIN {X 0,Y 587.631,Z 480.575,A -85,B 0,C 180,E1 -1518.583,E2 -1518.583} C_VEL
LIN {X 0,Y 587.532,Z 492.62,A -85,B 0,C 180,E1 -1519.14,E2 -1519.14} C_VEL
LIN {X 0,Y 587.467,Z 504.193,A -85,B 0,C 180,E1 -1519.836,E2 -1519.836} C_VEL
LIN {X 0,Y 587.392,Z 514.59,A -85,B 0,C 180,E1 -1520.617,E2 -1520.617} C_VEL
LIN {X 0,Y 587.322,Z 523.106,A -85,B 0,C 180,E1 -1521.397,E2 -1521.397} C_VEL
LIN {X 0,Y 587.274,Z 530.955,A -85,B 0,C 180,E1 -1522.262,E2 -1522.262} C_VEL
LIN {X 0,Y 587.231,Z 537.465,A -85,B 0,C 180,E1 -1523.126,E2 -1523.126} C_VEL
LIN {X 0,Y 587.236,Z 543.863,A -85,B 0,C 180,E1 -1524.161,E2 -1524.161} C_VEL
LIN {X 0,Y 587.147,Z 548.947,A -85,B 0,C 180,E1 -1525.193,E2 -1525.193} C_VEL
LIN {X 0,Y 587.212,Z 552.894,A -85,B 0,C 180,E1 -1526.225,E2 -1526.225} C_VEL
LIN {X 0,Y 587.132,Z 555.808,A -85,B 0,C 180,E1 -1527.255,E2 -1527.255} C_VEL
LIN {X 0,Y 587.141,Z 557.2,A -85,B 0,C 180,E1 -1527.941,E2 -1527.941} C_VEL
LIN {X 0,Y 587.14,Z 558.784,A -85,B 0,C 180,E1 -1529.313,E2 -1529.313} C_VEL
LIN {X 0,Y 587.137,Z 559,A -85,B 0,C 180,E1 -1529.999,E2 -1529.999} C_VEL
LIN {X 0,Y 587.147,Z 558.186,A -85,B 0,C 180,E1 -1531.371,E2 -1531.371} C_VEL
LIN {X 0,Y 587.141,Z 557.201,A -85,B 0,C 180,E1 -1532.057,E2 -1532.057} C_VEL
LIN {X 0,Y 587.132,Z 555.81,A -85,B 0,C 180,E1 -1532.744,E2 -1532.744} C_VEL
LIN {X 0,Y 587.212,Z 552.898,A -85,B 0,C 180,E1 -1533.774,E2 -1533.774} C_VEL
LIN {X 0,Y 587.147,Z 548.953,A -85,B 0,C 180,E1 -1534.806,E2 -1534.806} C_VEL
LIN {X 0,Y 587.217,Z 542.881,A -85,B 0,C 180,E1 -1536.01,E2 -1536.01} C_VEL
LIN {X 0,Y 587.244,Z 536.242,A -85,B 0,C 180,E1 -1537.045,E2 -1537.045} C_VEL
LIN {X 0,Y 587.299,Z 527.996,A -85,B 0,C 180,E1 -1538.082,E2 -1538.082} C_VEL
LIN {X 0,Y 587.343,Z 519.546,A -85,B 0,C 180,E1 -1538.948,E2 -1538.948} C_VEL
LIN {X 0,Y 587.418,Z 509.106,A -85,B 0,C 180,E1 -1539.816,E2 -1539.816} C_VEL
LIN {X 0,Y 587.488,Z 498.769,A -85,B 0,C 180,E1 -1540.511,E2 -1540.511} C_VEL
LIN {X 0,Y 587.582,Z 486.824,A -85,B 0,C 180,E1 -1541.148,E2 -1541.148} C_VEL
LIN {X 0,Y 587.627,Z 474.62,A -85,B 0,C 180,E1 -1541.639,E2 -1541.639} C_VEL
LIN {X 0,Y 587.703,Z 461.471,A -85,B 0,C 180,E1 -1542.013,E2 -1542.013} C_VEL
LIN {X 0,Y 587.775,Z 449.141,A -85,B 0,C 180,E1 -1542.231,E2 -1542.231} C_VEL
LIN {X 0,Y 587.726,Z 348.547,A -85,B 0,C 180,E1 -1543.467,E2 -1543.467} C_VEL
LIN {X 0,Y 587.409,Z 346.278,A -85,B 0,C 180,E1 -1543.535,E2 -1543.535} C_VEL
LIN {X 0,Y 587.55,Z 325.337,A -85,B 0,C 180,E1 -1546.325,E2 -1546.325} C_VEL
LIN {X 0,Y 587.735,Z 302.409,A -85,B 0,C 180,E1 -1549.423,E2 -1549.423} C_VEL
LIN {X 0,Y 587.893,Z 280.131,A -85,B 0,C 180,E1 -1552.491,E2 -1552.491} C_VEL
LIN {X 0,Y 587.823,Z 274.812,A -85,B 0,C 180,E1 -1553.237,E2 -1553.237} C_VEL
LIN {X 0,Y 587.328,Z 272.326,A -85,B 0,C 180,E1 -1553.631,E2 -1553.631} C_VEL
LIN {X 0,Y 587.327,Z 272.328,A -85,B 0,C 180,E1 -1556.278,E2 -1556.278} C_VEL
LIN {X 0,Y 587.343,Z 272.318,A -85,B 0,C 180,E1 -1559.132,E2 -1559.132} C_VEL
LIN {X 0,Y 587.337,Z 272.326,A -85,B 0,C 180,E1 -1561.834,E2 -1561.834} C_VEL
LIN {X 0,Y 587.338,Z 272.321,A -85,B 0,C 180,E1 -1564.346,E2 -1564.346} C_VEL
LIN {X 0,Y 587.337,Z 272.324,A -85,B 0,C 180,E1 -1567.607,E2 -1567.607} C_VEL
LIN {X 0,Y 587.304,Z 272.325,A -85,B 0,C 180,E1 -1570.254,E2 -1570.254} C_VEL
LIN {X 0,Y 587.296,Z 272.325,A -85,B 0,C 180,E1 -1573.116,E2 -1573.116} C_VEL
LIN {X 0,Y 587.292,Z 272.327,A -85,B 0,C 180,E1 -1576.046,E2 -1576.046} C_VEL
LIN {X 0,Y 587.324,Z 272.321,A -85,B 0,C 180,E1 -1578.925,E2 -1578.925} C_VEL
LIN {X 0,Y 587.31,Z 272.331,A -85,B 0,C 180,E1 -1581.519,E2 -1581.519} C_VEL
LIN {X 0,Y 587.281,Z 272.326,A -85,B 0,C 180,E1 -1584.099,E2 -1584.099} C_VEL
LIN {X 0,Y 587.327,Z 272.323,A -85,B 0,C 180,E1 -1586.888,E2 -1586.888} C_VEL
LIN {X 0,Y 587.311,Z 272.328,A -85,B 0,C 180,E1 -1589.493,E2 -1589.493} C_VEL
LIN {X 0,Y 587.295,Z 272.331,A -85,B 0,C 180,E1 -1591.401,E2 -1591.401} C_VEL
LIN {X 0,Y 587.286,Z 272.326,A -85,B 0,C 180,E1 -1593.831,E2 -1593.831} C_VEL
LIN {X 0,Y 587.289,Z 272.329,A -85,B 0,C 180,E1 -1596.74,E2 -1596.74} C_VEL
LIN {X 0,Y 587.301,Z 272.324,A -85,B 0,C 180,E1 -1599.694,E2 -1599.694} C_VEL
LIN {X 0,Y 587.274,Z 272.326,A -85,B 0,C 180,E1 -1601.872,E2 -1601.872} C_VEL
LIN {X 0,Y 587.29,Z 272.325,A -85,B 0,C 180,E1 -1604.024,E2 -1604.024} C_VEL
LIN {X 0,Y 587.278,Z 272.336,A -85,B 0,C 180,E1 -1606.857,E2 -1606.857} C_VEL
LIN {X 0,Y 587.327,Z 272.326,A -85,B 0,C 180,E1 -1608.962,E2 -1608.962} C_VEL
LIN {X 0,Y 587.298,Z 272.323,A -85,B 0,C 180,E1 -1611.744,E2 -1611.744} C_VEL
LIN {X 0,Y 587.334,Z 272.327,A -85,B 0,C 180,E1 -1614.507,E2 -1614.507} C_VEL
LIN {X 0,Y 587.327,Z 272.321,A -85,B 0,C 180,E1 -1617.257,E2 -1617.257} C_VEL
LIN {X 0,Y 587.346,Z 272.32,A -85,B 0,C 180,E1 -1620,E2 -1620} C_VEL
LIN {X 0,Y 587.35,Z 272.321,A -85,B 0,C 180,E1 -1622.743,E2 -1622.743} C_VEL
LIN {X 0,Y 587.31,Z 272.322,A -85,B 0,C 180,E1 -1625.493,E2 -1625.493} C_VEL
LIN {X 0,Y 587.311,Z 272.331,A -85,B 0,C 180,E1 -1628.256,E2 -1628.256} C_VEL
LIN {X 0,Y 587.321,Z 272.321,A -85,B 0,C 180,E1 -1631.125,E2 -1631.125} C_VEL
LIN {X 0,Y 587.337,Z 272.324,A -85,B 0,C 180,E1 -1633.846,E2 -1633.846} C_VEL
LIN {X 0,Y 587.316,Z 272.322,A -85,B 0,C 180,E1 -1636.807,E2 -1636.807} C_VEL
LIN {X 0,Y 587.284,Z 272.33,A -85,B 0,C 180,E1 -1638.308,E2 -1638.308} C_VEL
LIN {X 0,Y 586.642,Z 272.407,A -85,B 0,C 180,E1 -1638.88,E2 -1638.88} C_VEL
LIN {X 0,Y 583.825,Z 272.764,A -85,B 0,C 180,E1 -1639.809,E2 -1639.809} C_VEL
LIN {X 0,Y 581.422,Z 273.061,A -85,B 0,C 180,E1 -1640.556,E2 -1640.556} C_VEL
LIN {X 0,Y 580.369,Z 273.189,A -85,B 0,C 180,E1 -1641.132,E2 -1641.132} C_VEL
LIN {X 0,Y 580.273,Z 273.2,A -85,B 0,C 180,E1 -1641.327,E2 -1641.327} C_VEL
LIN {X 0,Y 580.289,Z 273.2,A -85,B 0,C 180,E1 -1644.317,E2 -1644.317} C_VEL
LIN {X 0,Y 580.247,Z 273.206,A -85,B 0,C 180,E1 -1647.404,E2 -1647.404} C_VEL
LIN {X 0,Y 580.276,Z 273.207,A -85,B 0,C 180,E1 -1649.774,E2 -1649.774} C_VEL
LIN {X 0,Y 580.286,Z 273.199,A -85,B 0,C 180,E1 -1652.202,E2 -1652.202} C_VEL
LIN {X 0,Y 580.278,Z 273.198,A -85,B 0,C 180,E1 -1654.697,E2 -1654.697} C_VEL
LIN {X 0,Y 580.28,Z 273.204,A -85,B 0,C 180,E1 -1657.27,E2 -1657.27} C_VEL
LIN {X 0,Y 580.281,Z 273.198,A -85,B 0,C 180,E1 -1660.271,E2 -1660.271} C_VEL
LIN {X 0,Y 580.254,Z 273.202,A -85,B 0,C 180,E1 -1662.709,E2 -1662.709} C_VEL
LIN {X 0,Y 580.258,Z 273.205,A -85,B 0,C 180,E1 -1665.611,E2 -1665.611} C_VEL
LIN {X 0,Y 580.274,Z 273.199,A -85,B 0,C 180,E1 -1668.232,E2 -1668.232} C_VEL
LIN {X 0,Y 580.271,Z 273.206,A -85,B 0,C 180,E1 -1670.966,E2 -1670.966} C_VEL
LIN {X 0,Y 580.264,Z 273.202,A -85,B 0,C 180,E1 -1673.597,E2 -1673.597} C_VEL
LIN {X 0,Y 580.276,Z 273.199,A -85,B 0,C 180,E1 -1676.144,E2 -1676.144} C_VEL
LIN {X 0,Y 580.27,Z 273.204,A -85,B 0,C 180,E1 -1678.615,E2 -1678.615} C_VEL
LIN {X 0,Y 580.289,Z 273.204,A -85,B 0,C 180,E1 -1681.025,E2 -1681.025} C_VEL
LIN {X 0,Y 580.288,Z 273.197,A -85,B 0,C 180,E1 -1683.668,E2 -1683.668} C_VEL
LIN {X 0,Y 580.294,Z 273.196,A -85,B 0,C 180,E1 -1685.684,E2 -1685.684} C_VEL
LIN {X 0,Y 580.27,Z 273.2,A -85,B 0,C 180,E1 -1687.948,E2 -1687.948} C_VEL
LIN {X 0,Y 580.3,Z 273.201,A -85,B 0,C 180,E1 -1690.914,E2 -1690.914} C_VEL
LIN {X 0,Y 580.304,Z 273.376,A -85,B 0,C 180,E1 -1691.738,E2 -1691.738} C_VEL
LIN {X 0,Y 580.351,Z 284.623,A -85,B 0,C 180,E1 -1693.828,E2 -1693.828} C_VEL
LIN {X 0,Y 580.312,Z 298.559,A -85,B 0,C 180,E1 -1696.385,E2 -1696.385} C_VEL
LIN {X 0,Y 580.99,Z 304.325,A -85,B 0,C 180,E1 -1696.491,E2 -1696.491} C_VEL
LIN {X 0,Y 580.801,Z 404.9,A -85,B 0,C 180,E1 -1697.753,E2 -1697.753} C_VEL
LIN {X 0,Y 580.741,Z 418.265,A -85,B 0,C 180,E1 -1698.062,E2 -1698.062} C_VEL
LIN {X 0,Y 580.664,Z 430.399,A -85,B 0,C 180,E1 -1698.481,E2 -1698.481} C_VEL
LIN {X 0,Y 580.558,Z 441.78,A -85,B 0,C 180,E1 -1699.009,E2 -1699.009} C_VEL
LIN {X 0,Y 580.47,Z 453.575,A -85,B 0,C 180,E1 -1699.713,E2 -1699.713} C_VEL
LIN {X 0,Y 580.344,Z 464.076,A -85,B 0,C 180,E1 -1700.504,E2 -1700.504} C_VEL
LIN {X 0,Y 580.301,Z 474.39,A -85,B 0,C 180,E1 -1701.469,E2 -1701.469} C_VEL
LIN {X 0,Y 580.199,Z 483.357,A -85,B 0,C 180,E1 -1702.519,E2 -1702.519} C_VEL
LIN {X 0,Y 580.135,Z 491.002,A -85,B 0,C 180,E1 -1703.637,E2 -1703.637} C_VEL
LIN {X 0,Y 580.085,Z 497.168,A -85,B 0,C 180,E1 -1704.787,E2 -1704.787} C_VEL
LIN {X 0,Y 580.105,Z 501.524,A -85,B 0,C 180,E1 -1705.832,E2 -1705.832} C_VEL
LIN {X 0,Y 580.123,Z 503.825,A -85,B 0,C 180,E1 -1706.528,E2 -1706.528} C_VEL
LIN {X 0,Y 580.043,Z 505.695,A -85,B 0,C 180,E1 -1707.223,E2 -1707.223} C_VEL
LIN {X 0,Y 580.04,Z 507.129,A -85,B 0,C 180,E1 -1707.918,E2 -1707.918} C_VEL
LIN {X 0,Y 580.04,Z 508.754,A -85,B 0,C 180,E1 -1709.306,E2 -1709.306} C_VEL
LIN {X 0,Y 580.038,Z 508.996,A -85,B 0,C 180,E1 -1710.001,E2 -1710.001} C_VEL
LIN {X 0,Y 580.04,Z 508.814,A -85,B 0,C 180,E1 -1710.695,E2 -1710.695} C_VEL
LIN {X 0,Y 580.04,Z 507.27,A -85,B 0,C 180,E1 -1712.084,E2 -1712.084} C_VEL
LIN {X 0,Y 580.044,Z 505.911,A -85,B 0,C 180,E1 -1712.779,E2 -1712.779} C_VEL
LIN {X 0,Y 580.11,Z 503.037,A -85,B 0,C 180,E1 -1713.821,E2 -1713.821} C_VEL
LIN {X 0,Y 580.054,Z 499.138,A -85,B 0,C 180,E1 -1714.866,E2 -1714.866} C_VEL
LIN {X 0,Y 580.162,Z 494.106,A -85,B 0,C 180,E1 -1715.911,E2 -1715.911} C_VEL
LIN {X 0,Y 580.185,Z 486.561,A -85,B 0,C 180,E1 -1717.133,E2 -1717.133} C_VEL
LIN {X 0,Y 580.246,Z 478.379,A -85,B 0,C 180,E1 -1718.183,E2 -1718.183} C_VEL
LIN {X 0,Y 580.308,Z 469.994,A -85,B 0,C 180,E1 -1719.059,E2 -1719.059} C_VEL
LIN {X 0,Y 580.421,Z 459.69,A -85,B 0,C 180,E1 -1719.936,E2 -1719.936} C_VEL
LIN {X 0,Y 580.499,Z 448.063,A -85,B 0,C 180,E1 -1720.728,E2 -1720.728} C_VEL
LIN {X 0,Y 580.623,Z 436.361,A -85,B 0,C 180,E1 -1721.349,E2 -1721.349} C_VEL
LIN {X 0,Y 580.673,Z 424.637,A -85,B 0,C 180,E1 -1721.826,E2 -1721.826} C_VEL
LIN {X 0,Y 580.784,Z 411.473,A -85,B 0,C 180,E1 -1722.204,E2 -1722.204} C_VEL
LIN {X 0,Y 580.862,Z 399.084,A -85,B 0,C 180,E1 -1722.424,E2 -1722.424} C_VEL
LIN {X 0,Y 580.931,Z 302.49,A -85,B 0,C 180,E1 -1723.623,E2 -1723.623} C_VEL
LIN {X 0,Y 580.293,Z 298.556,A -85,B 0,C 180,E1 -1723.706,E2 -1723.706} C_VEL
LIN {X 0,Y 580.389,Z 283.146,A -85,B 0,C 180,E1 -1726.533,E2 -1726.533} C_VEL
LIN {X 0,Y 580.287,Z 273.2,A -85,B 0,C 180,E1 -1728.401,E2 -1728.401} C_VEL
LIN {X 0,Y 580.29,Z 273.204,A -85,B 0,C 180,E1 -1731.306,E2 -1731.306} C_VEL
LIN {X 0,Y 580.276,Z 273.206,A -85,B 0,C 180,E1 -1733.559,E2 -1733.559} C_VEL
LIN {X 0,Y 580.283,Z 273.2,A -85,B 0,C 180,E1 -1735.85,E2 -1735.85} C_VEL
LIN {X 0,Y 580.301,Z 273.195,A -85,B 0,C 180,E1 -1738.186,E2 -1738.186} C_VEL
LIN {X 0,Y 580.277,Z 273.2,A -85,B 0,C 180,E1 -1740.693,E2 -1740.693} C_VEL
LIN {X 0,Y 580.289,Z 273.206,A -85,B 0,C 180,E1 -1743.314,E2 -1743.314} C_VEL
LIN {X 0,Y 580.248,Z 273.204,A -85,B 0,C 180,E1 -1745.756,E2 -1745.756} C_VEL
LIN {X 0,Y 580.289,Z 273.196,A -85,B 0,C 180,E1 -1748.147,E2 -1748.147} C_VEL
LIN {X 0,Y 580.301,Z 273.201,A -85,B 0,C 180,E1 -1750.844,E2 -1750.844} C_VEL
LIN {X 0,Y 580.284,Z 273.199,A -85,B 0,C 180,E1 -1753.658,E2 -1753.658} C_VEL
LIN {X 0,Y 580.278,Z 273.201,A -85,B 0,C 180,E1 -1756.61,E2 -1756.61} C_VEL
LIN {X 0,Y 580.302,Z 273.202,A -85,B 0,C 180,E1 -1759.157,E2 -1759.157} C_VEL
LIN {X 0,Y 580.292,Z 273.196,A -85,B 0,C 180,E1 -1761.927,E2 -1761.927} C_VEL
LIN {X 0,Y 580.255,Z 273.204,A -85,B 0,C 180,E1 -1764.453,E2 -1764.453} C_VEL
LIN {X 0,Y 580.292,Z 273.204,A -85,B 0,C 180,E1 -1766.975,E2 -1766.975} C_VEL
LIN {X 0,Y 580.299,Z 273.196,A -85,B 0,C 180,E1 -1769.425,E2 -1769.425} C_VEL
LIN {X 0,Y 580.293,Z 273.197,A -85,B 0,C 180,E1 -1772.143,E2 -1772.143} C_VEL
LIN {X 0,Y 580.326,Z 273.193,A -85,B 0,C 180,E1 -1775.27,E2 -1775.27} C_VEL
LIN {X 0,Y 580.273,Z 273.199,A -85,B 0,C 180,E1 -1777.947,E2 -1777.947} C_VEL
LIN {X 0,Y 580.298,Z 273.203,A -85,B 0,C 180,E1 -1780.913,E2 -1780.913} C_VEL
LIN {X 0,Y 580.326,Z 273.371,A -85,B 0,C 180,E1 -1781.738,E2 -1781.738} C_VEL
LIN {X 0,Y 580.345,Z 284.618,A -85,B 0,C 180,E1 -1783.827,E2 -1783.827} C_VEL
LIN {X 0,Y 580.314,Z 298.893,A -85,B 0,C 180,E1 -1786.407,E2 -1786.407} C_VEL
LIN {X 0,Y 580.951,Z 304.254,A -85,B 0,C 180,E1 -1786.489,E2 -1786.489} C_VEL
LIN {X 0,Y 580.758,Z 404.713,A -85,B 0,C 180,E1 -1787.751,E2 -1787.751} C_VEL
LIN {X 0,Y 580.763,Z 418.241,A -85,B 0,C 180,E1 -1788.062,E2 -1788.062} C_VEL
LIN {X 0,Y 580.668,Z 430.317,A -85,B 0,C 180,E1 -1788.481,E2 -1788.481} C_VEL
LIN {X 0,Y 580.564,Z 441.709,A -85,B 0,C 180,E1 -1789.009,E2 -1789.009} C_VEL
LIN {X 0,Y 580.443,Z 453.564,A -85,B 0,C 180,E1 -1789.712,E2 -1789.712} C_VEL
LIN {X 0,Y 580.342,Z 464.064,A -85,B 0,C 180,E1 -1790.503,E2 -1790.503} C_VEL
LIN {X 0,Y 580.272,Z 472.644,A -85,B 0,C 180,E1 -1791.292,E2 -1791.292} C_VEL
LIN {X 0,Y 580.222,Z 480.543,A -85,B 0,C 180,E1 -1792.168,E2 -1792.168} C_VEL
LIN {X 0,Y 580.164,Z 487.119,A -85,B 0,C 180,E1 -1793.042,E2 -1793.042} C_VEL
LIN {X 0,Y 580.167,Z 493.579,A -85,B 0,C 180,E1 -1794.09,E2 -1794.09} C_VEL
LIN {X 0,Y 580.052,Z 498.729,A -85,B 0,C 180,E1 -1795.135,E2 -1795.135} C_VEL
LIN {X 0,Y 580.11,Z 502.725,A -85,B 0,C 180,E1 -1796.179,E2 -1796.179} C_VEL
LIN {X 0,Y 580.043,Z 505.682,A -85,B 0,C 180,E1 -1797.222,E2 -1797.222} C_VEL
LIN {X 0,Y 580.047,Z 508.138,A -85,B 0,C 180,E1 -1798.611,E2 -1798.611} C_VEL
LIN {X 0,Y 580.041,Z 508.753,A -85,B 0,C 180,E1 -1799.306,E2 -1799.306} C_VEL
LIN {X 0,Y 580.04,Z 508.812,A -85,B 0,C 180,E1 -1800.694,E2 -1800.694} C_VEL
LIN {X 0,Y 580.047,Z 508.24,A -85,B 0,C 180,E1 -1801.389,E2 -1801.389} C_VEL
LIN {X 0,Y 580.044,Z 505.909,A -85,B 0,C 180,E1 -1802.778,E2 -1802.778} C_VEL
LIN {X 0,Y 580.11,Z 503.038,A -85,B 0,C 180,E1 -1803.821,E2 -1803.821} C_VEL
LIN {X 0,Y 580.054,Z 499.136,A -85,B 0,C 180,E1 -1804.865,E2 -1804.865} C_VEL
LIN {X 0,Y 580.161,Z 494.084,A -85,B 0,C 180,E1 -1805.91,E2 -1805.91} C_VEL
LIN {X 0,Y 580.158,Z 487.731,A -85,B 0,C 180,E1 -1806.958,E2 -1806.958} C_VEL
LIN {X 0,Y 580.241,Z 479.856,A -85,B 0,C 180,E1 -1808.007,E2 -1808.007} C_VEL
LIN {X 0,Y 580.308,Z 470.013,A -85,B 0,C 180,E1 -1809.058,E2 -1809.058} C_VEL
LIN {X 0,Y 580.415,Z 459.659,A -85,B 0,C 180,E1 -1809.936,E2 -1809.936} C_VEL
LIN {X 0,Y 580.504,Z 449.417,A -85,B 0,C 180,E1 -1810.639,E2 -1810.639} C_VEL
LIN {X 0,Y 580.592,Z 438.185,A -85,B 0,C 180,E1 -1811.261,E2 -1811.261} C_VEL
LIN {X 0,Y 580.667,Z 425.764,A -85,B 0,C 180,E1 -1811.785,E2 -1811.785} C_VEL
LIN {X 0,Y 580.733,Z 413.19,A -85,B 0,C 180,E1 -1812.16,E2 -1812.16} C_VEL
LIN {X 0,Y 580.824,Z 400.643,A -85,B 0,C 180,E1 -1812.402,E2 -1812.402} C_VEL
LIN {X 0,Y 580.937,Z 302.538,A -85,B 0,C 180,E1 -1813.623,E2 -1813.623} C_VEL
LIN {X 0,Y 580.31,Z 298.559,A -85,B 0,C 180,E1 -1813.705,E2 -1813.705} C_VEL
LIN {X 0,Y 580.383,Z 283.149,A -85,B 0,C 180,E1 -1816.533,E2 -1816.533} C_VEL
LIN {X 0,Y 580.275,Z 273.242,A -85,B 0,C 180,E1 -1818.378,E2 -1818.378} C_VEL
LIN {X 0,Y 580.278,Z 273.207,A -85,B 0,C 180,E1 -1821.306,E2 -1821.306} C_VEL
LIN {X 0,Y 580.247,Z 273.208,A -85,B 0,C 180,E1 -1823.559,E2 -1823.559} C_VEL
LIN {X 0,Y 580.253,Z 273.202,A -85,B 0,C 180,E1 -1826.325,E2 -1826.325} C_VEL
LIN {X 0,Y 580.247,Z 273.209,A -85,B 0,C 180,E1 -1829.299,E2 -1829.299} C_VEL
LIN {X 0,Y 580.27,Z 273.2,A -85,B 0,C 180,E1 -1832.202,E2 -1832.202} C_VEL
LIN {X 0,Y 580.268,Z 273.206,A -85,B 0,C 180,E1 -1834.698,E2 -1834.698} C_VEL
LIN {X 0,Y 580.261,Z 273.203,A -85,B 0,C 180,E1 -1837.271,E2 -1837.271} C_VEL
LIN {X 0,Y 580.279,Z 273.201,A -85,B 0,C 180,E1 -1840.268,E2 -1840.268} C_VEL
LIN {X 0,Y 580.234,Z 273.204,A -85,B 0,C 180,E1 -1843.385,E2 -1843.385} C_VEL
LIN {X 0,Y 580.23,Z 273.211,A -85,B 0,C 180,E1 -1846.337,E2 -1846.337} C_VEL
LIN {X 0,Y 580.259,Z 273.201,A -85,B 0,C 180,E1 -1849.153,E2 -1849.153} C_VEL
LIN {X 0,Y 580.281,Z 273.202,A -85,B 0,C 180,E1 -1851.929,E2 -1851.929} C_VEL
LIN {X 0,Y 580.233,Z 273.21,A -85,B 0,C 180,E1 -1854.451,E2 -1854.451} C_VEL
LIN {X 0,Y 580.29,Z 273.198,A -85,B 0,C 180,E1 -1856.975,E2 -1856.975} C_VEL
LIN {X 0,Y 580.285,Z 273.2,A -85,B 0,C 180,E1 -1859.424,E2 -1859.424} C_VEL
LIN {X 0,Y 580.26,Z 273.208,A -85,B 0,C 180,E1 -1862.149,E2 -1862.149} C_VEL
LIN {X 0,Y 580.326,Z 273.196,A -85,B 0,C 180,E1 -1865.27,E2 -1865.27} C_VEL
LIN {X 0,Y 580.293,Z 273.279,A -85,B 0,C 180,E1 -1866.253,E2 -1866.253} C_VEL
LIN {X 0,Y 580.988,Z 278.177,A -85,B 0,C 180,E1 -1866.953,E2 -1866.953} C_VEL
LIN {X 0,Y 580.833,Z 296.075,A -85,B 0,C 180,E1 -1869.457,E2 -1869.457} C_VEL
LIN {X 0,Y 580.622,Z 317.349,A -85,B 0,C 180,E1 -1872.385,E2 -1872.385} C_VEL
LIN {X 0,Y 580.474,Z 338.622,A -85,B 0,C 180,E1 -1875.27,E2 -1875.27} C_VEL
LIN {X 0,Y 580.4,Z 346.517,A -85,B 0,C 180,E1 -1876.33,E2 -1876.33} C_VEL
LIN {X 0,Y 580.99,Z 352.458,A -85,B 0,C 180,E1 -1876.423,E2 -1876.423} C_VEL
LIN {X 0,Y 580.805,Z 454.912,A -85,B 0,C 180,E1 -1877.707,E2 -1877.707} C_VEL
LIN {X 0,Y 580.739,Z 468.192,A -85,B 0,C 180,E1 -1878.016,E2 -1878.016} C_VEL
LIN {X 0,Y 580.664,Z 479.858,A -85,B 0,C 180,E1 -1878.416,E2 -1878.416} C_VEL
LIN {X 0,Y 580.586,Z 490.918,A -85,B 0,C 180,E1 -1878.92,E2 -1878.92} C_VEL
LIN {X 0,Y 580.48,Z 501.576,A -85,B 0,C 180,E1 -1879.536,E2 -1879.536} C_VEL
LIN {X 0,Y 580.375,Z 512.465,A -85,B 0,C 180,E1 -1880.327,E2 -1880.327} C_VEL
LIN {X 0,Y 580.272,Z 523.106,A -85,B 0,C 180,E1 -1881.292,E2 -1881.292} C_VEL
LIN {X 0,Y 580.222,Z 530.955,A -85,B 0,C 180,E1 -1882.167,E2 -1882.167} C_VEL
LIN {X 0,Y 580.154,Z 538.648,A -85,B 0,C 180,E1 -1883.221,E2 -1883.221} C_VEL
LIN {X 0,Y 580.139,Z 545.676,A -85,B 0,C 180,E1 -1884.438,E2 -1884.438} C_VEL
LIN {X 0,Y 580.108,Z 550.369,A -85,B 0,C 180,E1 -1885.483,E2 -1885.483} C_VEL
LIN {X 0,Y 580.123,Z 553.956,A -85,B 0,C 180,E1 -1886.527,E2 -1886.527} C_VEL
LIN {X 0,Y 580.043,Z 555.808,A -85,B 0,C 180,E1 -1887.221,E2 -1887.221} C_VEL
LIN {X 0,Y 580.04,Z 557.199,A -85,B 0,C 180,E1 -1887.916,E2 -1887.916} C_VEL
LIN {X 0,Y 580.04,Z 558.784,A -85,B 0,C 180,E1 -1889.305,E2 -1889.305} C_VEL
LIN {X 0,Y 580.037,Z 559,A -85,B 0,C 180,E1 -1889.999,E2 -1889.999} C_VEL
LIN {X 0,Y 580.047,Z 558.186,A -85,B 0,C 180,E1 -1891.388,E2 -1891.388} C_VEL
LIN {X 0,Y 580.04,Z 557.2,A -85,B 0,C 180,E1 -1892.082,E2 -1892.082} C_VEL
LIN {X 0,Y 580.043,Z 555.81,A -85,B 0,C 180,E1 -1892.777,E2 -1892.777} C_VEL
LIN {X 0,Y 580.109,Z 552.898,A -85,B 0,C 180,E1 -1893.82,E2 -1893.82} C_VEL
LIN {X 0,Y 580.054,Z 548.953,A -85,B 0,C 180,E1 -1894.865,E2 -1894.865} C_VEL
LIN {X 0,Y 580.139,Z 542.881,A -85,B 0,C 180,E1 -1896.084,E2 -1896.084} C_VEL
LIN {X 0,Y 580.183,Z 536.243,A -85,B 0,C 180,E1 -1897.132,E2 -1897.132} C_VEL
LIN {X 0,Y 580.25,Z 527.997,A -85,B 0,C 180,E1 -1898.181,E2 -1898.181} C_VEL
LIN {X 0,Y 580.307,Z 519.546,A -85,B 0,C 180,E1 -1899.058,E2 -1899.058} C_VEL
LIN {X 0,Y 580.425,Z 509.108,A -85,B 0,C 180,E1 -1899.935,E2 -1899.935} C_VEL
LIN {X 0,Y 580.494,Z 498.767,A -85,B 0,C 180,E1 -1900.639,E2 -1900.639} C_VEL
LIN {X 0,Y 580.596,Z 487.254,A -85,B 0,C 180,E1 -1901.264,E2 -1901.264} C_VEL
LIN {X 0,Y 580.68,Z 474.5,A -85,B 0,C 180,E1 -1901.784,E2 -1901.784} C_VEL
LIN {X 0,Y 580.75,Z 461.47,A -85,B 0,C 180,E1 -1902.159,E2 -1902.159} C_VEL
LIN {X 0,Y 580.86,Z 449.141,A -85,B 0,C 180,E1 -1902.379,E2 -1902.379} C_VEL
LIN {X 0,Y 580.813,Z 349.22,A -85,B 0,C 180,E1 -1903.622,E2 -1903.622} C_VEL
LIN {X 0,Y 580.418,Z 346.445,A -85,B 0,C 180,E1 -1903.679,E2 -1903.679} C_VEL
LIN {X 0,Y 580.562,Z 325.337,A -85,B 0,C 180,E1 -1906.527,E2 -1906.527} C_VEL
LIN {X 0,Y 580.773,Z 303.751,A -85,B 0,C 180,E1 -1909.48,E2 -1909.48} C_VEL
LIN {X 0,Y 581.011,Z 281.46,A -85,B 0,C 180,E1 -1912.584,E2 -1912.584} C_VEL
LIN {X 0,Y 580.939,Z 276.456,A -85,B 0,C 180,E1 -1913.288,E2 -1913.288} C_VEL
LIN {X 0,Y 580.288,Z 273.205,A -85,B 0,C 180,E1 -1913.793,E2 -1913.793} C_VEL
LIN {X 0,Y 580.281,Z 273.205,A -85,B 0,C 180,E1 -1916.331,E2 -1916.331} C_VEL
LIN {X 0,Y 580.295,Z 273.197,A -85,B 0,C 180,E1 -1919.308,E2 -1919.308} C_VEL
LIN {X 0,Y 580.292,Z 273.202,A -85,B 0,C 180,E1 -1922.2,E2 -1922.2} C_VEL
LIN {X 0,Y 580.282,Z 273.197,A -85,B 0,C 180,E1 -1924.696,E2 -1924.696} C_VEL
LIN {X 0,Y 580.283,Z 273.199,A -85,B 0,C 180,E1 -1927.268,E2 -1927.268} C_VEL
LIN {X 0,Y 580.284,Z 273.199,A -85,B 0,C 180,E1 -1930.269,E2 -1930.269} C_VEL
LIN {X 0,Y 580.254,Z 273.201,A -85,B 0,C 180,E1 -1932.707,E2 -1932.707} C_VEL
LIN {X 0,Y 580.244,Z 273.211,A -85,B 0,C 180,E1 -1935.61,E2 -1935.61} C_VEL
LIN {X 0,Y 580.269,Z 273.2,A -85,B 0,C 180,E1 -1938.23,E2 -1938.23} C_VEL
LIN {X 0,Y 580.261,Z 273.202,A -85,B 0,C 180,E1 -1940.964,E2 -1940.964} C_VEL
LIN {X 0,Y 580.259,Z 273.207,A -85,B 0,C 180,E1 -1943.596,E2 -1943.596} C_VEL
LIN {X 0,Y 580.271,Z 273.199,A -85,B 0,C 180,E1 -1946.142,E2 -1946.142} C_VEL
LIN {X 0,Y 580.258,Z 273.201,A -85,B 0,C 180,E1 -1948.613,E2 -1948.613} C_VEL
LIN {X 0,Y 580.276,Z 273.205,A -85,B 0,C 180,E1 -1951.023,E2 -1951.023} C_VEL
LIN {X 0,Y 580.246,Z 273.204,A -85,B 0,C 180,E1 -1953.673,E2 -1953.673} C_VEL
LIN {X 0,Y 580.239,Z 273.204,A -85,B 0,C 180,E1 -1956.44,E2 -1956.44} C_VEL
LIN {X 0,Y 580.253,Z 273.204,A -85,B 0,C 180,E1 -1959.436,E2 -1959.436} C_VEL
LIN {X 0,Y 580.236,Z 273.204,A -85,B 0,C 180,E1 -1961.644,E2 -1961.644} C_VEL
LIN {X 0,Y 580.241,Z 273.203,A -85,B 0,C 180,E1 -1963.824,E2 -1963.824} C_VEL
LIN {X 0,Y 580.235,Z 273.211,A -85,B 0,C 180,E1 -1966.695,E2 -1966.695} C_VEL
LIN {X 0,Y 580.296,Z 273.205,A -85,B 0,C 180,E1 -1968.827,E2 -1968.827} C_VEL
LIN {X 0,Y 580.273,Z 273.199,A -85,B 0,C 180,E1 -1971.643,E2 -1971.643} C_VEL
LIN {X 0,Y 580.297,Z 273.203,A -85,B 0,C 180,E1 -1974.44,E2 -1974.44} C_VEL
LIN {X 0,Y 580.297,Z 273.197,A -85,B 0,C 180,E1 -1977.223,E2 -1977.223} C_VEL
LIN {X 0,Y 580.317,Z 273.196,A -85,B 0,C 180,E1 -1980,E2 -1980} C_VEL
LIN {X 0,Y 580.314,Z 273.198,A -85,B 0,C 180,E1 -1982.777,E2 -1982.777} C_VEL
LIN {X 0,Y 580.279,Z 273.199,A -85,B 0,C 180,E1 -1985.56,E2 -1985.56} C_VEL
LIN {X 0,Y 580.283,Z 273.206,A -85,B 0,C 180,E1 -1988.357,E2 -1988.357} C_VEL
LIN {X 0,Y 580.292,Z 273.196,A -85,B 0,C 180,E1 -1991.191,E2 -1991.191} C_VEL
LIN {X 0,Y 580.299,Z 273.204,A -85,B 0,C 180,E1 -1994.018,E2 -1994.018} C_VEL
LIN {X 0,Y 580.281,Z 273.198,A -85,B 0,C 180,E1 -1996.907,E2 -1996.907} C_VEL
LIN {X 0,Y 580.269,Z 273.207,A -85,B 0,C 180,E1 -1999.824,E2 -1999.824} C_VEL
LIN {X 0,Y 580.273,Z 273.2,A -85,B 0,C 180,E1 -2001.327,E2 -2001.327} C_VEL
LIN {X 0,Y 579.572,Z 273.295,A -85,B 0,C 180,E1 -2001.907,E2 -2001.907} C_VEL
LIN {X 0,Y 576.694,Z 273.65,A -85,B 0,C 180,E1 -2002.846,E2 -2002.846} C_VEL
LIN {X 0,Y 574.301,Z 273.949,A -85,B 0,C 180,E1 -2003.603,E2 -2003.603} C_VEL
